KUKA KRL program: MyProgram_101().src

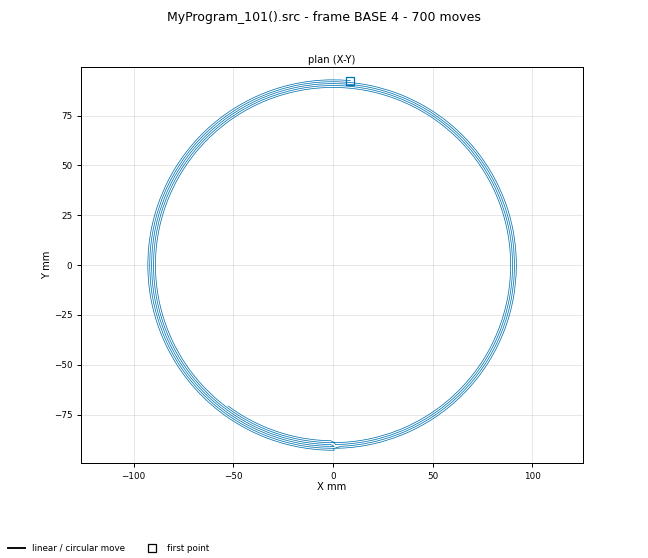
[picture p0: tool path of MyProgram_101().src in frame BASE 4, 700 of 700 moves have a stored position in this frame; points joined in program order, loops and branches not executed]
&ACCESS RVP
&REL 1
&PARAM TEMPLATE = C:\KRC\Roboter\Template\vorgabe
&PARAM EDITMASK = *
DEF MyProgram_101()
; ---- Setting reference (Base) ----
$BASE = BASE_DATA[4]

; --------------------------
; ---- Setting tool (TCP) ----
$TOOL = TOOL_DATA[3]
; --------------------------

$VEL.CP = VEL_APROX_PRINT
Startdeposition()
$VEL.CP = VEL_PRINT
LIN {X 8.6685,Y 92.5128,Z 92,A 80.0856,B 24.9063,C -2.2344,E1 25.0131,E2 4.9435} C_DIS
LIN {X 3.5626,Y 92.8506,Z 92,A 82.8753,B 24.9074,C -2.2219,E1 25.0054,E2 2.1844} C_DIS
LIN {X -2.3592,Y 92.8893,Z 92,A 87.6518,B 24.9042,C -2.2593,E1 24.9918,E2 -2.6809} C_DIS
LIN {X -7.3293,Y 92.6285,Z 92,A 89.5483,B 24.9077,C -2.2184,E1 24.9868,E2 -4.481} C_DIS
LIN {X -9.3778,Y 92.444,Z 92,A 91.7647,B 24.9051,C -2.2495,E1 24.9805,E2 -6.7727} C_DIS
LIN {X -13.6164,Y 91.9165,Z 92,A 93.6976,B 24.9072,C -2.2243,E1 24.9753,E2 -8.6472} C_DIS
LIN {X -16.7897,Y 91.3891,Z 92,A 95.4705,B 24.9079,C -2.2159,E1 24.9704,E2 -10.4018} C_DIS
LIN {X -20.8381,Y 90.5513,Z 92,A 98.1416,B 24.9077,C -2.2177,E1 24.9631,E2 -13.0804} C_DIS
LIN {X -24.0491,Y 89.752,Z 92,A 100.1644,B 24.908,C -2.2151,E1 24.9577,E2 -15.1} C_DIS
LIN {X -27.0285,Y 88.9015,Z 92,A 102.8086,B 24.9061,C -2.2371,E1 24.9504,E2 -17.8011} C_DIS
LIN {X -30.6581,Y 87.7146,Z 92,A 104.1863,B 24.909,C -2.2023,E1 24.947,E2 -19.0985} C_DIS
LIN {X -35.7226,Y 85.7771,Z 92,A 108.0632,B 24.908,C -2.215,E1 24.9368,E2 -23.0141} C_DIS
LIN {X -39.4719,Y 84.1178,Z 92,A 110.5653,B 24.9084,C -2.2103,E1 24.9305,E2 -25.5112} C_DIS
LIN {X -43.093,Y 82.3213,Z 92,A 112.9702,B 24.9089,C -2.2035,E1 24.9245,E2 -27.9061} C_DIS
LIN {X -46.2813,Y 80.5717,Z 92,A 115.1055,B 24.9095,C -2.1961,E1 24.9193,E2 -30.0302} C_DIS
LIN {X -49.1228,Y 78.8715,Z 92,A 116.9389,B 24.9104,C -2.1857,E1 24.915,E2 -31.8445} C_DIS
LIN {X -51.7549,Y 77.1709,Z 92,A 119.2261,B 24.9098,C -2.1933,E1 24.9096,E2 -34.1572} C_DIS
LIN {X -54.5832,Y 75.1969,Z 92,A 121.3196,B 24.9102,C -2.188,E1 24.9049,E2 -36.2452} C_DIS
LIN {X -57.0235,Y 73.3636,Z 92,A 123.1994,B 24.9105,C -2.1839,E1 24.9007,E2 -38.1223} C_DIS
LIN {X -59.5641,Y 71.3156,Z 92,A 124.9102,B 24.9117,C -2.17,E1 24.8971,E2 -39.8064} C_DIS
LIN {X -62.1969,Y 69.0317,Z 92,A 127.4401,B 24.9111,C -2.1772,E1 24.8917,E2 -42.3633} C_DIS
LIN {X -64.7695,Y 66.6245,Z 92,A 129.5058,B 24.9118,C -2.1687,E1 24.8876,E2 -44.4172} C_DIS
LIN {X -66.9884,Y 64.392,Z 92,A 131.5448,B 24.9119,C -2.167,E1 24.8836,E2 -46.4612} C_DIS
LIN {X -68.5485,Y 62.7286,Z 92,A 133.1466,B 24.9117,C -2.1697,E1 24.8805,E2 -48.0763} C_DIS
LIN {X -71.3556,Y 59.516,Z 92,A 135.5018,B 24.913,C -2.1543,E1 24.8763,E2 -50.4056} C_DIS
LIN {X -73.2264,Y 57.2008,Z 92,A 137.5086,B 24.913,C -2.1548,E1 24.8728,E2 -52.423} C_DIS
LIN {X -75.6618,Y 53.9356,Z 92,A 140.3542,B 24.9126,C -2.1585,E1 24.8681,E2 -55.2912} C_DIS
LIN {X -78.3706,Y 49.919,Z 92,A 143.006,B 24.9141,C -2.1396,E1 24.8641,E2 -57.9114} C_DIS
LIN {X -79.8357,Y 47.5405,Z 92,A 145.45,B 24.9127,C -2.1573,E1 24.8605,E2 -60.4101} C_DIS
LIN {X -81.9789,Y 43.7432,Z 92,A 147.2305,B 24.9156,C -2.1211,E1 24.8583,E2 -62.1138} C_DIS
LIN {X -83.9639,Y 39.7993,Z 92,A 150.1955,B 24.9156,C -2.1205,E1 24.8546,E2 -65.0933} C_DIS
LIN {X -86.8415,Y 33.0503,Z 92,A 155.4811,B 24.9149,C -2.1304,E1 24.849,E2 -70.4321} C_DIS
LIN {X -88.3197,Y 28.8698,Z 92,A 157.4147,B 24.9175,C -2.0971,E1 24.8473,E2 -72.297} C_DIS
LIN {X -89.2816,Y 25.7437,Z 92,A 159.2439,B 24.9185,C -2.085,E1 24.8459,E2 -74.1079} C_DIS
LIN {X -90.3116,Y 21.8542,Z 92,A 161.8727,B 24.9187,C -2.0817,E1 24.844,E2 -76.7442} C_DIS
LIN {X -91.0374,Y 18.5998,Z 92,A 163.664,B 24.9199,C -2.0671,E1 24.843,E2 -78.5112} C_DIS
LIN {X -91.5949,Y 15.6278,Z 92,A 166.1987,B 24.9187,C -2.0817,E1 24.8417,E2 -81.0959} C_DIS
LIN {X -92.2271,Y 11.3219,Z 92,A 168.754,B 24.9197,C -2.0691,E1 24.8408,E2 -83.6364} C_DIS
LIN {X -92.6128,Y 7.5252,Z 92,A 171.2761,B 24.9199,C -2.0668,E1 24.8401,E2 -86.1681} C_DIS
LIN {X -92.9096,Y 1.2732,Z 92,A 175.048,B 24.9211,C -2.0517,E1 24.8398,E2 -89.9267} C_DIS
LIN {X -92.8996,Y -1.852,Z 92,A 177.8358,B 24.9195,C -2.0723,E1 24.84,E2 -92.7805} C_DIS
LIN {X -92.65,Y -7.0609,Z 92,A -179.9339,B 24.9226,C -2.0314,E1 24.8404,E2 -94.9264} C_DIS
LIN {X -92.3349,Y -10.401,Z 92,A -177.8054,B 24.923,C -2.0267,E1 24.841,E2 -97.0564} C_DIS
LIN {X -91.8721,Y -13.905,Z 92,A -175.6926,B 24.9237,C -2.0178,E1 24.8418,E2 -99.1606} C_DIS
LIN {X -91.3402,Y -17.0584,Z 92,A -173.6234,B 24.9239,C -2.0146,E1 24.8428,E2 -101.2346} C_DIS
LIN {X -90.635,Y -20.4756,Z 92,A -171.7293,B 24.925,C -2,E1 24.8439,E2 -103.105} C_DIS
LIN {X -89.8976,Y -23.5016,Z 92,A -168.9165,B 24.9233,C -2.022,E1 24.8459,E2 -105.9866} C_DIS
LIN {X -88.8201,Y -27.2909,Z 92,A -167.1243,B 24.9254,C -1.9947,E1 24.8473,E2 -107.7241} C_DIS
LIN {X -87.6746,Y -30.7721,Z 92,A -164.9819,B 24.9262,C -1.9844,E1 24.8492,E2 -109.854} C_DIS
LIN {X -86.4825,Y -33.9783,Z 92,A -162.2464,B 24.9252,C -1.9979,E1 24.852,E2 -112.6371} C_DIS
LIN {X -85.1973,Y -37.0834,Z 92,A -160.6883,B 24.9268,C -1.9758,E1 24.8537,E2 -114.1511} C_DIS
LIN {X -83.8317,Y -40.0753,Z 92,A -158.6212,B 24.9271,C -1.9713,E1 24.8562,E2 -116.2188} C_DIS
LIN {X -82.2602,Y -43.2091,Z 92,A -156.425,B 24.9275,C -1.9664,E1 24.859,E2 -118.4152} C_DIS
LIN {X -79.7757,Y -47.6421,Z 92,A -153.2654,B 24.9281,C -1.9589,E1 24.8633,E2 -121.5731} C_DIS
LIN {X -77.3395,Y -51.5028,Z 92,A -150.4483,B 24.9286,C -1.9517,E1 24.8676,E2 -124.3874} C_DIS
LIN {X -74.9207,Y -54.9604,Z 92,A -147.9325,B 24.9293,C -1.9425,E1 24.8717,E2 -126.8935} C_DIS
LIN {X -72.9573,Y -57.5411,Z 92,A -145.9634,B 24.9297,C -1.9367,E1 24.875,E2 -128.8583} C_DIS
LIN {X -70.924,Y -60.0302,Z 92,A -143.3889,B 24.9286,C -1.9511,E1 24.8797,E2 -131.4788} C_DIS
LIN {X -68.7858,Y -62.47,Z 92,A -141.7905,B 24.9299,C -1.9337,E1 24.8826,E2 -133.0429} C_DIS
LIN {X -67.1259,Y -64.2492,Z 92,A -139.9944,B 24.9294,C -1.94,E1 24.8861,E2 -134.8618} C_DIS
LIN {X -63.1282,Y -68.1818,Z 92,A -136.838,B 24.9307,C -1.9231,E1 24.8924,E2 -137.991} C_DIS
LIN {X -60.9567,Y -70.1291,Z 92,A -135.1059,B 24.9311,C -1.9175,E1 24.8961,E2 -139.7165} C_DIS
LIN {X -58.2775,Y -72.3711,Z 92,A -132.4598,B 24.9302,C -1.9295,E1 24.9019,E2 -142.4012} C_DIS
LIN {X -54.9904,Y -74.8987,Z 92,A -130.2116,B 24.9313,C -1.9149,E1 24.9068,E2 -144.6228} C_DIS
LIN {X -51.8971,Y -77.0746,Z 92,A -128.2718,B 24.9324,C -1.8983,E1 24.9112,E2 -146.5296} C_DIS
LIN {X -49.5179,Y -78.6247,Z 92,A -126.3962,B 24.9324,C -1.8996,E1 24.9156,E2 -148.4145} C_DIS
LIN {X -44.9776,Y -81.3062,Z 92,A -122.7756,B 24.9318,C -1.9072,E1 24.9245,E2 -152.0639} C_DIS
LIN {X -40.832,Y -83.467,Z 92,A -119.7997,B 24.9318,C -1.9067,E1 24.9319,E2 -155.0464} C_DIS
LIN {X -36.8853,Y -85.2837,Z 92,A -117.4804,B 24.9329,C -1.8918,E1 24.9377,E2 -157.3359} C_DIS
LIN {X -33.9003,Y -86.5132,Z 92,A -115.3671,B 24.9328,C -1.8939,E1 24.9432,E2 -159.4589} C_DIS
LIN {X -30.6688,Y -87.7108,Z 92,A -112.9272,B 24.9321,C -1.9027,E1 24.9497,E2 -161.9245} C_DIS
LIN {X -26.0912,Y -89.1803,Z 92,A -110.4074,B 24.9334,C -1.8855,E1 24.9563,E2 -164.4077} C_DIS
LIN {X -22.9049,Y -90.0509,Z 92,A -107.9771,B 24.9325,C -1.8976,E1 24.963,E2 -166.8706} C_DIS
LIN {X -18.0534,Y -91.1486,Z 92,A -105.1442,B 24.9332,C -1.8882,E1 24.9707,E2 -169.6846} C_DIS
LIN {X -12.8895,Y -92.0198,Z 92,A -102.102,B 24.9337,C -1.8809,E1 24.979,E2 -172.7123} C_DIS
LIN {X -8.1132,Y -92.5641,Z 92,A -98.9097,B 24.9331,C -1.8884,E1 24.9879,E2 -175.9242} C_DIS
LIN {X -5.2842,Y -92.7677,Z 92,A -96.7874,B 24.9322,C -1.9014,E1 24.9939,E2 -178.0781} C_DIS
LIN {X -2.0857,Y -92.8953,Z 92,A -95.1973,B 24.9332,C -1.8884,E1 24.9983,E2 -179.6373} C_DIS
LIN {X 0.616,Y -92.9061,Z 92,A -93.7308,B 24.9336,C -1.882,E1 25.0024,E2 -181.0887} C_DIS
Enddeposition()
LIN {X 0.616,Y -92.9061,Z 92,A -93.7308,B 24.9336,C -1.882,E1 25.0024,E2 -181.0887} C_DIS
Startdeposition()
$VEL.CP = VEL_PRINT
LIN {X 0.2828,Y -91.9616,Z 92,A -94.5574,B 24.9339,C -1.8772,E1 25,E2 -180.2507} C_DIS
LIN {X -5.5997,Y -91.7928,Z 92,A -98.2442,B 24.934,C -1.876,E1 24.9897,E2 -176.5604} C_DIS
LIN {X -11.5025,Y -91.2403,Z 92,A -102.7915,B 24.936,C -1.848,E1 24.9769,E2 -171.9441} C_DIS
LIN {X -15.3961,Y -90.6643,Z 92,A -104.5195,B 24.9343,C -1.8726,E1 24.9723,E2 -170.273} C_DIS
LIN {X -18.6363,Y -90.0539,Z 92,A -107.2484,B 24.9358,C -1.8513,E1 24.9647,E2 -167.4902} C_DIS
LIN {X -22.3727,Y -89.2006,Z 92,A -108.8615,B 24.9339,C -1.8779,E1 24.9605,E2 -165.9382} C_DIS
LIN {X -24.9821,Y -88.5037,Z 92,A -110.8484,B 24.9345,C -1.869,E1 24.955,E2 -163.927} C_DIS
LIN {X -27.644,Y -87.7097,Z 92,A -113.1828,B 24.9358,C -1.8507,E1 24.9487,E2 -161.545} C_DIS
LIN {X -31.573,Y -86.3721,Z 92,A -114.7673,B 24.9334,C -1.8854,E1 24.9448,E2 -160.0398} C_DIS
LIN {X -33.8196,Y -85.5177,Z 92,A -116.5155,B 24.9338,C -1.8786,E1 24.9401,E2 -158.2718} C_DIS
LIN {X -37.183,Y -84.1109,Z 92,A -119.0663,B 24.9343,C -1.872,E1 24.9335,E2 -155.6992} C_DIS
LIN {X -40.4944,Y -82.5672,Z 92,A -121.1125,B 24.9336,C -1.8821,E1 24.9284,E2 -153.6718} C_DIS
LIN {X -43.5278,Y -81.009,Z 92,A -123.807,B 24.9347,C -1.8667,E1 24.9217,E2 -150.9332} C_DIS
LIN {X -46.6784,Y -79.2347,Z 92,A -125.4312,B 24.933,C -1.8899,E1 24.9179,E2 -149.3592} C_DIS
LIN {X -48.8539,Y -77.9122,Z 92,A -127.4045,B 24.9337,C -1.8799,E1 24.9131,E2 -147.3561} C_DIS
LIN {X -51.7207,Y -76.0395,Z 92,A -129.5924,B 24.9337,C -1.8816,E1 24.9081,E2 -145.1649} C_DIS
LIN {X -55.1728,Y -73.5728,Z 92,A -132.7055,B 24.9343,C -1.8716,E1 24.901,E2 -142.0168} C_DIS
LIN {X -58.7179,Y -70.7758,Z 92,A -134.2641,B 24.9312,C -1.916,E1 24.8979,E2 -140.5582} C_DIS
LIN {X -60.4642,Y -69.2898,Z 92,A -136.1318,B 24.932,C -1.9049,E1 24.8938,E2 -138.6567} C_DIS
LIN {X -64.9463,Y -65.1083,Z 92,A -140.1141,B 24.9318,C -1.9076,E1 24.8858,E2 -134.6645} C_DIS
LIN {X -67.8507,Y -62.0749,Z 92,A -143.4197,B 24.9329,C -1.8922,E1 24.8794,E2 -131.3075} C_DIS
LIN {X -70.7868,Y -58.7047,Z 92,A -144.8676,B 24.9295,C -1.9398,E1 24.877,E2 -129.9665} C_DIS
LIN {X -73.1722,Y -55.7055,Z 92,A -148.3649,B 24.9315,C -1.9113,E1 24.8708,E2 -126.3846} C_DIS
LIN {X -75.2745,Y -52.8291,Z 92,A -149.7922,B 24.9294,C -1.9411,E1 24.8686,E2 -125.0214} C_DIS
LIN {X -76.6509,Y -50.8103,Z 92,A -152.1221,B 24.9309,C -1.9203,E1 24.8649,E2 -122.6302} C_DIS
LIN {X -78.5609,Y -47.8035,Z 92,A -154.4332,B 24.9307,C -1.9233,E1 24.8615,E2 -120.3145} C_DIS
LIN {X -80.5191,Y -44.4285,Z 92,A -155.9549,B 24.9282,C -1.9574,E1 24.8596,E2 -118.8662} C_DIS
LIN {X -82.2624,Y -41.1094,Z 92,A -158.5863,B 24.9284,C -1.9548,E1 24.8561,E2 -116.2145} C_DIS
LIN {X -83.5972,Y -38.3248,Z 92,A -160.6338,B 24.9282,C -1.9565,E1 24.8537,E2 -114.1598} C_DIS
LIN {X -85.0169,Y -35.0606,Z 92,A -163.1255,B 24.9284,C -1.9546,E1 24.851,E2 -111.6498} C_DIS
LIN {X -87.0622,Y -29.6179,Z 92,A -166.3552,B 24.9267,C -1.9771,E1 24.848,E2 -108.4554} C_DIS
LIN {X -88.9962,Y -23.1677,Z 92,A -170.3149,B 24.9252,C -1.9968,E1 24.8449,E2 -104.52} C_DIS
LIN {X -89.9931,Y -18.9325,Z 92,A -173.4017,B 24.9255,C -1.9938,E1 24.8429,E2 -101.4079} C_DIS
LIN {X -90.6389,Y -15.5479,Z 92,A -175.5804,B 24.925,C -1.9995,E1 24.8418,E2 -99.2299} C_DIS
LIN {X -91.1795,Y -11.9711,Z 92,A -177.8201,B 24.9245,C -2.007,E1 24.841,E2 -96.9948} C_DIS
LIN {X -91.5934,Y -8.2281,Z 92,A 179.8874,B 24.9238,C -2.0161,E1 24.8403,E2 -94.71} C_DIS
LIN {X -91.9262,Y -2.5761,Z 92,A 176.4109,B 24.9228,C -2.0288,E1 24.8398,E2 -91.2431} C_DIS
LIN {X -91.9611,Y 0.452,Z 92,A 173.6815,B 24.9243,C -2.0099,E1 24.8398,E2 -88.4521} C_DIS
LIN {X -91.8509,Y 4.5052,Z 92,A 171.9899,B 24.9218,C -2.0427,E1 24.84,E2 -86.8287} C_DIS
LIN {X -91.7204,Y 6.6768,Z 92,A 170.4237,B 24.9219,C -2.0407,E1 24.8403,E2 -85.2484} C_DIS
LIN {X -91.3851,Y 10.292,Z 92,A 168.0913,B 24.9215,C -2.0459,E1 24.841,E2 -82.9142} C_DIS
LIN {X -90.947,Y 13.6316,Z 92,A 165.9194,B 24.9212,C -2.0504,E1 24.8419,E2 -80.7403} C_DIS
LIN {X -90.2374,Y 17.7291,Z 92,A 163.7941,B 24.9194,C -2.0726,E1 24.8429,E2 -78.6551} C_DIS
LIN {X -89.3345,Y 21.8254,Z 92,A 159.9783,B 24.9216,C -2.0453,E1 24.8454,E2 -74.7518} C_DIS
LIN {X -88.1157,Y 26.3181,Z 92,A 158.5099,B 24.9175,C -2.0969,E1 24.8464,E2 -73.3981} C_DIS
LIN {X -85.8343,Y 33.0105,Z 92,A 153.8445,B 24.9171,C -2.1026,E1 24.8506,E2 -68.7199} C_DIS
LIN {X -83.9426,Y 37.5591,Z 92,A 150.096,B 24.918,C -2.0916,E1 24.8548,E2 -64.9242} C_DIS
LIN {X -81.4075,Y 42.7764,Z 92,A 146.5129,B 24.917,C -2.1032,E1 24.8593,E2 -61.3495} C_DIS
LIN {X -78.8588,Y 47.3134,Z 92,A 143.6783,B 24.9153,C -2.1247,E1 24.8632,E2 -58.5515} C_DIS
LIN {X -75.1466,Y 53.0116,Z 92,A 138.8684,B 24.9158,C -2.1193,E1 24.8707,E2 -53.7046} C_DIS
LIN {X -72.4594,Y 56.6294,Z 92,A 136.3327,B 24.9145,C -2.1349,E1 24.8749,E2 -51.1942} C_DIS
LIN {X -70.1399,Y 59.4763,Z 92,A 133.514,B 24.9153,C -2.1249,E1 24.88,E2 -48.3386} C_DIS
LIN {X -67.6898,Y 62.2503,Z 92,A 131.9427,B 24.9131,C -2.1529,E1 24.8829,E2 -46.827} C_DIS
LIN {X -65.6704,Y 64.3779,Z 92,A 129.8996,B 24.9132,C -2.1507,E1 24.8869,E2 -44.77} C_DIS
LIN {X -63.0701,Y 66.9266,Z 92,A 127.6993,B 24.9126,C -2.1582,E1 24.8913,E2 -42.5783} C_DIS
LIN {X -58.7476,Y 70.7511,Z 92,A 124.1726,B 24.9118,C -2.1684,E1 24.8987,E2 -39.0621} C_DIS
LIN {X -56.3635,Y 72.6652,Z 92,A 122.0966,B 24.9119,C -2.1672,E1 24.9032,E2 -36.9756} C_DIS
LIN {X -53.4043,Y 74.8664,Z 92,A 119.5836,B 24.9121,C -2.1653,E1 24.9089,E2 -34.4492} C_DIS
LIN {X -48.3848,Y 78.2053,Z 92,A 116.0419,B 24.9109,C -2.1791,E1 24.9172,E2 -30.9289} C_DIS
LIN {X -45.5415,Y 79.8941,Z 92,A 113.9873,B 24.9106,C -2.1829,E1 24.9221,E2 -28.8773} C_DIS
LIN {X -41.9369,Y 81.8432,Z 92,A 110.8076,B 24.9119,C -2.1677,E1 24.9301,E2 -25.6527} C_DIS
LIN {X -38.4781,Y 83.5258,Z 92,A 109.4852,B 24.9088,C -2.205,E1 24.9333,E2 -24.4156} C_DIS
LIN {X -32.1419,Y 86.1632,Z 92,A 104.9607,B 24.909,C -2.2031,E1 24.945,E2 -19.8763} C_DIS
LIN {X -26.3547,Y 88.1049,Z 92,A 101.0991,B 24.9087,C -2.2057,E1 24.9552,E2 -16.0139} C_DIS
LIN {X -23.8607,Y 88.8126,Z 92,A 99.4038,B 24.9088,C -2.2048,E1 24.9598,E2 -14.3139} C_DIS
LIN {X -19.4825,Y 89.8746,Z 92,A 96.4999,B 24.9088,C -2.2043,E1 24.9677,E2 -11.4049} C_DIS
LIN {X -16.833,Y 90.41,Z 92,A 94.7575,B 24.9089,C -2.2038,E1 24.9725,E2 -9.6592} C_DIS
LIN {X -13.905,Y 90.9047,Z 92,A 92.9109,B 24.9088,C -2.2052,E1 24.9776,E2 -7.8144} C_DIS
LIN {X -9.4125,Y 91.4791,Z 92,A 90.4784,B 24.9076,C -2.2195,E1 24.9842,E2 -5.414} C_DIS
LIN {X -7.0352,Y 91.6929,Z 92,A 87.9373,B 24.9104,C -2.1859,E1 24.9915,E2 -2.7923} C_DIS
LIN {X -2.9739,Y 91.9139,Z 92,A 86.3341,B 24.9078,C -2.217,E1 24.9958,E2 -1.2625} C_DIS
LIN {X 1.9013,Y 91.9425,Z 92,A 83.2214,B 24.908,C -2.2151,E1 25.0045,E2 1.8546} C_DIS
LIN {X 8.2335,Y 91.5929,Z 92,A 79.4639,B 24.9074,C -2.2215,E1 25.0149,E2 5.5954} C_DIS
LIN {X 12.3597,Y 91.1292,Z 92,A 76.4373,B 24.9087,C -2.2064,E1 25.0234,E2 8.6557} C_DIS
LIN {X 15.7547,Y 90.6039,Z 92,A 73.6994,B 24.9104,C -2.1858,E1 25.0311,E2 11.4394} C_DIS
LIN {X 19.649,Y 89.8383,Z 92,A 71.9868,B 24.9084,C -2.21,E1 25.0356,E2 13.0925} C_DIS
LIN {X 22.2254,Y 89.2369,Z 92,A 70.0924,B 24.9091,C -2.2008,E1 25.0408,E2 15.0061} C_DIS
LIN {X 28.415,Y 87.4619,Z 92,A 66.2333,B 24.909,C -2.203,E1 25.0511,E2 18.8531} C_DIS
LIN {X 31.8114,Y 86.2852,Z 92,A 63.9048,B 24.9094,C -2.198,E1 25.0572,E2 21.1888} C_DIS
LIN {X 34.3944,Y 85.2884,Z 92,A 61.9301,B 24.9102,C -2.1878,E1 25.0624,E2 23.1831} C_DIS
LIN {X 38.7426,Y 83.4027,Z 92,A 59.388,B 24.9093,C -2.1985,E1 25.0688,E2 25.6937} C_DIS
LIN {X 43.4952,Y 81.0255,Z 92,A 56.0505,B 24.9098,C -2.1933,E1 25.0771,E2 29.0342} C_DIS
LIN {X 46.2149,Y 79.5072,Z 92,A 53.7973,B 24.9109,C -2.1797,E1 25.0826,E2 31.3127} C_DIS
LIN {X 49.9134,Y 77.2381,Z 92,A 51.2644,B 24.9107,C -2.1815,E1 25.0885,E2 33.8334} C_DIS
LIN {X 52.3849,Y 75.5833,Z 92,A 49.0162,B 24.9121,C -2.1647,E1 25.0938,E2 36.1135} C_DIS
LIN {X 55.3268,Y 73.4571,Z 92,A 46.7079,B 24.9126,C -2.1591,E1 25.0989,E2 38.4268} C_DIS
LIN {X 58.3824,Y 71.0545,Z 92,A 45.1022,B 24.9106,C -2.1831,E1 25.1023,E2 39.9698} C_DIS
LIN {X 60.6518,Y 69.126,Z 92,A 43.0142,B 24.9116,C -2.1713,E1 25.1067,E2 42.0775} C_DIS
LIN {X 63.6497,Y 66.3759,Z 92,A 40.7956,B 24.9111,C -2.1773,E1 25.1112,E2 44.2728} C_DIS
LIN {X 65.3279,Y 64.7246,Z 92,A 39.0883,B 24.912,C -2.1657,E1 25.1146,E2 46.0004} C_DIS
LIN {X 68.0138,Y 61.8971,Z 92,A 36.3554,B 24.9133,C -2.1496,E1 25.1199,E2 48.7594} C_DIS
LIN {X 70.6202,Y 58.905,Z 92,A 34.2149,B 24.9128,C -2.1556,E1 25.1237,E2 50.8758} C_DIS
LIN {X 73.0518,Y 55.8618,Z 92,A 32.0135,B 24.9127,C -2.1579,E1 25.1275,E2 53.0615} C_DIS
LIN {X 74.5764,Y 53.8107,Z 92,A 29.9752,B 24.9143,C -2.138,E1 25.1309,E2 55.137} C_DIS
LIN {X 77.6741,Y 49.2342,Z 92,A 26.6174,B 24.9147,C -2.1322,E1 25.1361,E2 58.4917} C_DIS
LIN {X 79.6578,Y 45.9528,Z 92,A 24.4327,B 24.9147,C -2.1332,E1 25.1391,E2 60.6628} C_DIS
LIN {X 81.5998,Y 42.4112,Z 92,A 21.7393,B 24.9157,C -2.12,E1 25.1427,E2 63.3733} C_DIS
LIN {X 83.0177,Y 39.562,Z 92,A 19.7845,B 24.9161,C -2.1154,E1 25.1451,E2 65.3283} C_DIS
LIN {X 85.2013,Y 34.6083,Z 92,A 16.157,B 24.9176,C -2.0966,E1 25.1491,E2 68.9804} C_DIS
LIN {X 86.6592,Y 30.7781,Z 92,A 14.0219,B 24.917,C -2.1042,E1 25.1511,E2 71.0856} C_DIS
LIN {X 87.8023,Y 27.3453,Z 92,A 11.6532,B 24.9178,C -2.0933,E1 25.1531,E2 73.4666} C_DIS
LIN {X 88.6607,Y 24.4231,Z 92,A 9.9022,B 24.9178,C -2.0929,E1 25.1545,E2 75.2086} C_DIS
LIN {X 89.8415,Y 19.634,Z 92,A 6.2087,B 24.9204,C -2.0609,E1 25.1568,E2 78.9561} C_DIS
LIN {X 90.6181,Y 15.6721,Z 92,A 4.555,B 24.9185,C -2.0844,E1 25.1576,E2 80.5446} C_DIS
LIN {X 91.4737,Y 9.4642,Z 92,A 0.6816,B 24.9194,C -2.0732,E1 25.159,E2 84.4215} C_DIS
LIN {X 91.8931,Y 3.5759,Z 92,A -2.9164,B 24.9201,C -2.0644,E1 25.1597,E2 88.019} C_DIS
LIN {X 91.9585,Y -0.8351,Z 92,A -5.8986,B 24.9214,C -2.047,E1 25.1597,E2 91.0245} C_DIS
LIN {X 91.8212,Y -5.0846,Z 92,A -8.9068,B 24.9231,C -2.0254,E1 25.1594,E2 94.0658} C_DIS
LIN {X 91.0208,Y -13.1238,Z 92,A -13.9681,B 24.9244,C -2.0082,E1 25.1577,E2 99.1377} C_DIS
LIN {X 90.5052,Y -16.3037,Z 92,A -15.455,B 24.9234,C -2.0208,E1 25.157,E2 100.5861} C_DIS
LIN {X 89.5013,Y -21.1332,Z 92,A -18.4839,B 24.924,C -2.0127,E1 25.1553,E2 103.6167} C_DIS
LIN {X 88.4836,Y -25.053,Z 92,A -21.0539,B 24.9248,C -2.003,E1 25.1534,E2 106.1947} C_DIS
LIN {X 87.4607,Y -28.4189,Z 92,A -23.724,B 24.9266,C -1.9787,E1 25.1511,E2 108.9071} C_DIS
LIN {X 86.3759,Y -31.5628,Z 92,A -24.797,B 24.9243,C -2.0089,E1 25.1502,E2 109.9028} C_DIS
LIN {X 85.1636,Y -34.701,Z 92,A -27.7218,B 24.9271,C -1.972,E1 25.1471,E2 112.8983} C_DIS
LIN {X 83.6955,Y -38.1075,Z 92,A -29.7485,B 24.9268,C -1.9754,E1 25.1448,E2 114.9061} C_DIS
LIN {X 81.3991,Y -42.7923,Z 92,A -32.6428,B 24.9266,C -1.9788,E1 25.1413,E2 117.777} C_DIS
LIN {X 79.0732,Y -46.9517,Z 92,A -35.8269,B 24.9278,C -1.9623,E1 25.1368,E2 120.9834} C_DIS
LIN {X 77.3233,Y -49.7808,Z 92,A -37.8365,B 24.9281,C -1.9587,E1 25.1338,E2 122.9914} C_DIS
LIN {X 75.5907,Y -52.3742,Z 92,A -39.8359,B 24.9286,C -1.9513,E1 25.1307,E2 124.9985} C_DIS
LIN {X 73.5566,Y -55.1944,Z 92,A -42.5624,B 24.9305,C -1.9251,E1 25.1261,E2 127.7736} C_DIS
LIN {X 71.339,Y -58.0325,Z 92,A -44.9739,B 24.9314,C -1.9132,E1 25.1218,E2 130.202} C_DIS
LIN {X 68.6019,Y -61.2437,Z 92,A -46.4496,B 24.9289,C -1.9481,E1 25.1193,E2 131.5888} C_DIS
LIN {X 66.9912,Y -63.0014,Z 92,A -49.0653,B 24.9321,C -1.9037,E1 25.1141,E2 134.2979} C_DIS
LIN {X 64.0171,Y -66.0218,Z 92,A -51.6536,B 24.9324,C -1.8992,E1 25.1089,E2 136.886} C_DIS
LIN {X 60.9981,Y -68.8217,Z 92,A -53.3271,B 24.9305,C -1.9251,E1 25.1056,E2 138.4916} C_DIS
LIN {X 59.1259,Y -70.4368,Z 92,A -55.7994,B 24.9331,C -1.8884,E1 25.1001,E2 141.041} C_DIS
LIN {X 55.7736,Y -73.1198,Z 92,A -58.1721,B 24.9328,C -1.8934,E1 25.0949,E2 143.3933} C_DIS
LIN {X 53.1514,Y -75.0468,Z 92,A -59.5537,B 24.9315,C -1.9122,E1 25.0919,E2 144.7257} C_DIS
LIN {X 50.879,Y -76.6056,Z 92,A -61.4423,B 24.9321,C -1.9027,E1 25.0875,E2 146.6304} C_DIS
LIN {X 48.0906,Y -78.3864,Z 92,A -63.8762,B 24.9333,C -1.8856,E1 25.0816,E2 149.0969} C_DIS
LIN {X 44.6891,Y -80.3735,Z 92,A -65.7662,B 24.9322,C -1.9011,E1 25.0771,E2 150.9445} C_DIS
LIN {X 42.1864,Y -81.7156,Z 92,A -68.261,B 24.9343,C -1.8726,E1 25.0708,E2 153.4998} C_DIS
LIN {X 38.955,Y -83.3038,Z 92,A -70.3855,B 24.9343,C -1.8733,E1 25.0654,E2 155.6174} C_DIS
LIN {X 35.9751,Y -84.6337,Z 92,A -71.6419,B 24.9325,C -1.8974,E1 25.0624,E2 156.8136} C_DIS
LIN {X 30.368,Y -86.8032,Z 92,A -75.9565,B 24.9343,C -1.8725,E1 25.051,E2 161.1779} C_DIS
LIN {X 24.4935,Y -88.6416,Z 92,A -79.3437,B 24.9335,C -1.8836,E1 25.042,E2 164.5328} C_DIS
LIN {X 20.2855,Y -89.6977,Z 92,A -82.3055,B 24.9343,C -1.872,E1 25.0339,E2 167.5178} C_DIS
LIN {X 16.8181,Y -90.4126,Z 92,A -84.2959,B 24.9339,C -1.8776,E1 25.0285,E2 169.4927} C_DIS
LIN {X 13.945,Y -90.8985,Z 92,A -86.7745,B 24.9356,C -1.8536,E1 25.0215,E2 172.0256} C_DIS
LIN {X 10.4021,Y -91.3722,Z 92,A -88.3174,B 24.9341,C -1.8755,E1 25.0174,E2 173.5154} C_DIS
LIN {X 5.3436,Y -91.8069,Z 92,A -91.2893,B 24.9337,C -1.8805,E1 25.0092,E2 176.474} C_DIS
LIN {X 0.5912,Y -91.9536,Z 92,A -93.06,B 24.9309,C -1.9205,E1 25.0046,E2 178.1492} C_DIS
Enddeposition()
LIN {X 0.5912,Y -91.9536,Z 92,A -93.06,B 24.9309,C -1.9205,E1 25.0046,E2 178.1492} C_DIS
Startdeposition()
$VEL.CP = VEL_PRINT
LIN {X 4.0889,Y -90.9141,Z 92,A -91.4298,B 24.931,C -1.9178,E1 25.009,E2 176.5259} C_DIS
LIN {X 7.1118,Y -90.7277,Z 92,A -89.5434,B 24.931,C -1.918,E1 25.0143,E2 174.64} C_DIS
LIN {X 11.0267,Y -90.3358,Z 92,A -86.7492,B 24.9301,C -1.9304,E1 25.0221,E2 171.8184} C_DIS
LIN {X 15.4148,Y -89.6918,Z 92,A -84.224,B 24.9307,C -1.9232,E1 25.029,E2 169.3128} C_DIS
LIN {X 18.7307,Y -89.0585,Z 92,A -81.8883,B 24.93,C -1.9323,E1 25.0354,E2 166.9583} C_DIS
LIN {X 22.6976,Y -88.1299,Z 92,A -79.7337,B 24.9308,C -1.9206,E1 25.0412,E2 164.8347} C_DIS
LIN {X 28.3671,Y -86.4726,Z 92,A -76.0286,B 24.9306,C -1.9243,E1 25.0511,E2 161.1274} C_DIS
LIN {X 33.2291,Y -84.7224,Z 92,A -72.5336,B 24.9297,C -1.9371,E1 25.0603,E2 157.6094} C_DIS
LIN {X 35.9929,Y -83.5867,Z 92,A -69.4735,B 24.9264,C -1.9819,E1 25.0684,E2 154.4506} C_DIS
LIN {X 41.4959,Y -80.9948,Z 92,A -66.8827,B 24.9292,C -1.9438,E1 25.0746,E2 151.957} C_DIS
LIN {X 43.7943,Y -79.7768,Z 92,A -64.4746,B 24.9269,C -1.9742,E1 25.0807,E2 149.484} C_DIS
LIN {X 47.7526,Y -77.4729,Z 92,A -62.381,B 24.9286,C -1.9511,E1 25.0855,E2 147.4514} C_DIS
LIN {X 50.6673,Y -75.5981,Z 92,A -60.2052,B 24.9283,C -1.9552,E1 25.0906,E2 145.2733} C_DIS
LIN {X 53.3211,Y -73.7511,Z 92,A -57.9909,B 24.9275,C -1.9658,E1 25.0957,E2 143.0416} C_DIS
LIN {X 57.8514,Y -70.2527,Z 92,A -54.6385,B 24.9276,C -1.9645,E1 25.103,E2 139.7046} C_DIS
LIN {X 60.4872,Y -67.9959,Z 92,A -52.6353,B 24.9278,C -1.963,E1 25.1072,E2 137.713} C_DIS
LIN {X 63.6055,Y -65.0896,Z 92,A -49.341,B 24.9256,C -1.9915,E1 25.1139,E2 134.365} C_DIS
LIN {X 65.9276,Y -62.7368,Z 92,A -47.6882,B 24.9264,C -1.981,E1 25.1171,E2 132.7441} C_DIS
LIN {X 68.2977,Y -60.1468,Z 92,A -45.8094,B 24.9269,C -1.9746,E1 25.1205,E2 130.8887} C_DIS
LIN {X 70.792,Y -57.189,Z 92,A -42.7931,B 24.9248,C -2.0021,E1 25.126,E2 127.8214} C_DIS
LIN {X 73.647,Y -53.4633,Z 92,A -40.1528,B 24.9251,C -1.9986,E1 25.1304,E2 125.202} C_DIS
LIN {X 75.6072,Y -50.6538,Z 92,A -37.9548,B 24.9245,C -2.0061,E1 25.1338,E2 122.9973} C_DIS
LIN {X 77.5721,Y -47.5898,Z 92,A -35.9516,B 24.9248,C -2.002,E1 25.1368,E2 121.0138} C_DIS
LIN {X 78.7192,Y -45.6671,Z 92,A -33.7958,B 24.9225,C -2.0336,E1 25.1399,E2 118.7946} C_DIS
LIN {X 80.4573,Y -42.5288,Z 92,A -31.4886,B 24.9218,C -2.042,E1 25.1429,E2 116.4796} C_DIS
LIN {X 82.1938,Y -39.069,Z 92,A -29.7158,B 24.9231,C -2.0247,E1 25.145,E2 114.7571} C_DIS
LIN {X 83.2065,Y -36.8648,Z 92,A -27.1306,B 24.9198,C -2.0686,E1 25.148,E2 112.0826} C_DIS
LIN {X 85.192,Y -32.0069,Z 92,A -25.5174,B 24.9238,C -2.0162,E1 25.1495,E2 110.602} C_DIS
LIN {X 86.69,Y -27.6951,Z 92,A -22.0075,B 24.9213,C -2.0484,E1 25.1527,E2 107.0358} C_DIS
LIN {X 87.432,Y -25.2574,Z 92,A -20.0533,B 24.9199,C -2.0663,E1 25.1543,E2 105.0505} C_DIS
LIN {X 88.373,Y -21.7325,Z 92,A -17.6187,B 24.919,C -2.0787,E1 25.1559,E2 102.6006} C_DIS
LIN {X 89.1538,Y -18.2665,Z 92,A -15.9697,B 24.9201,C -2.064,E1 25.1568,E2 100.996} C_DIS
LIN {X 89.6825,Y -15.4705,Z 92,A -13.9298,B 24.9189,C -2.0789,E1 25.1578,E2 98.9328} C_DIS
LIN {X 90.5655,Y -8.9565,Z 92,A -10.0396,B 24.9186,C -2.083,E1 25.1592,E2 95.056} C_DIS
LIN {X 90.7781,Y -6.442,Z 92,A -7.8966,B 24.9166,C -2.1087,E1 25.1596,E2 92.8651} C_DIS
LIN {X 90.9629,Y -2.7958,Z 92,A -6.198,B 24.9178,C -2.0938,E1 25.1598,E2 91.2118} C_DIS
LIN {X 90.9773,Y 2.328,Z 92,A -2.945,B 24.9169,C -2.1051,E1 25.1597,E2 87.9515} C_DIS
LIN {X 90.6145,Y 8.4312,Z 92,A 0.3099,B 24.9176,C -2.0955,E1 25.1591,E2 84.7384} C_DIS
LIN {X 90.1396,Y 12.5298,Z 92,A 3.3549,B 24.9157,C -2.1201,E1 25.1581,E2 81.6535} C_DIS
LIN {X 89.6348,Y 15.7419,Z 92,A 5.1777,B 24.9158,C -2.1182,E1 25.1573,E2 79.8458} C_DIS
LIN {X 88.8806,Y 19.5531,Z 92,A 8.1185,B 24.9138,C -2.144,E1 25.1556,E2 76.8613} C_DIS
LIN {X 87.8792,Y 23.6498,Z 92,A 10.4875,B 24.914,C -2.1416,E1 25.1539,E2 74.5117} C_DIS
LIN {X 86.5175,Y 28.2284,Z 92,A 13.5636,B 24.9131,C -2.1531,E1 25.1514,E2 71.4259} C_DIS
LIN {X 85.6258,Y 30.829,Z 92,A 15.9552,B 24.9107,C -2.1825,E1 25.1491,E2 68.9784} C_DIS
LIN {X 84.1007,Y 34.7763,Z 92,A 18.5421,B 24.9103,C -2.1873,E1 25.1463,E2 66.3943} C_DIS
LIN {X 82.5188,Y 38.3759,Z 92,A 20.2715,B 24.9119,C -2.167,E1 25.1444,E2 64.7222} C_DIS
LIN {X 81.2799,Y 40.9382,Z 92,A 22.5783,B 24.91,C -2.1907,E1 25.1414,E2 62.3717} C_DIS
LIN {X 79.7525,Y 43.839,Z 92,A 24.2243,B 24.9108,C -2.1811,E1 25.1393,E2 60.757} C_DIS
LIN {X 78.0224,Y 46.8488,Z 92,A 26.1366,B 24.9111,C -2.177,E1 25.1366,E2 58.8642} C_DIS
LIN {X 76.6997,Y 48.9822,Z 92,A 27.8851,B 24.9103,C -2.1872,E1 25.134,E2 57.1004} C_DIS
LIN {X 74.1284,Y 52.7926,Z 92,A 30.7477,B 24.9098,C -2.1934,E1 25.1295,E2 54.2373} C_DIS
LIN {X 72.0309,Y 55.6203,Z 92,A 32.7592,B 24.9099,C -2.1914,E1 25.1261,E2 52.2401} C_DIS
LIN {X 70.2232,Y 57.887,Z 92,A 34.8185,B 24.9089,C -2.2041,E1 25.1224,E2 50.1603} C_DIS
LIN {X 67.8811,Y 60.6155,Z 92,A 37.616,B 24.9068,C -2.2284,E1 25.1172,E2 47.318} C_DIS
LIN {X 65.4345,Y 63.2487,Z 92,A 39.2331,B 24.9084,C -2.2102,E1 25.1142,E2 45.7509} C_DIS
LIN {X 63.6182,Y 65.077,Z 92,A 41.173,B 24.9071,C -2.2249,E1 25.1102,E2 43.7844} C_DIS
LIN {X 60.8933,Y 67.6324,Z 92,A 43.3793,B 24.9071,C -2.2245,E1 25.1057,E2 41.588} C_DIS
LIN {X 57.7897,Y 70.304,Z 92,A 46.1511,B 24.9062,C -2.2362,E1 25.0997,E2 38.7991} C_DIS
LIN {X 51.6912,Y 74.9011,Z 92,A 50.4513,B 24.907,C -2.2267,E1 25.0902,E2 34.5368} C_DIS
LIN {X 48.399,Y 77.0691,Z 92,A 52.9909,B 24.9065,C -2.2326,E1 25.0842,E2 31.9915} C_DIS
LIN {X 45.4085,Y 78.8679,Z 92,A 55.2063,B 24.9062,C -2.2364,E1 25.0789,E2 29.7738} C_DIS
LIN {X 40.5775,Y 81.4589,Z 92,A 58.6855,B 24.9057,C -2.2419,E1 25.0703,E2 26.2915} C_DIS
LIN {X 37.5743,Y 82.8872,Z 92,A 60.7616,B 24.9056,C -2.2437,E1 25.065,E2 24.2163} C_DIS
LIN {X 35.3703,Y 83.8511,Z 92,A 62.4322,B 24.905,C -2.2507,E1 25.0607,E2 22.5331} C_DIS
LIN {X 29.8783,Y 85.9618,Z 92,A 65.6623,B 24.906,C -2.238,E1 25.0524,E2 19.3401} C_DIS
LIN {X 24.1516,Y 87.7437,Z 92,A 69.8729,B 24.9046,C -2.2555,E1 25.041,E2 15.0956} C_DIS
LIN {X 20.8164,Y 88.5938,Z 92,A 71.6754,B 24.9055,C -2.2444,E1 25.0362,E2 13.322} C_DIS
LIN {X 16.0231,Y 89.5842,Z 92,A 74.9716,B 24.9048,C -2.2529,E1 25.0271,E2 10.0095} C_DIS
LIN {X 12.7202,Y 90.1125,Z 92,A 77.0283,B 24.9048,C -2.2519,E1 25.0215,E2 7.9572} C_DIS
LIN {X 8.7069,Y 90.589,Z 92,A 79.4111,B 24.9053,C -2.2469,E1 25.0149,E2 5.5879} C_DIS
LIN {X 3.7103,Y 90.9304,Z 92,A 82.9071,B 24.9043,C -2.2582,E1 25.0051,E2 2.0664} C_DIS
LIN {X 0.1571,Y 91.0066,Z 92,A 85.1596,B 24.9043,C -2.2584,E1 24.9988,E2 -0.1862} C_DIS
LIN {X -3.6061,Y 90.9348,Z 92,A 87.8918,B 24.9034,C -2.2696,E1 24.9911,E2 -2.9455} C_DIS
LIN {X -6.8065,Y 90.7521,Z 92,A 89.5196,B 24.9045,C -2.2559,E1 24.9866,E2 -4.5414} C_DIS
LIN {X -10.0755,Y 90.4478,Z 92,A 91.3556,B 24.9053,C -2.2473,E1 24.9816,E2 -6.358} C_DIS
LIN {X -13.6589,Y 89.9753,Z 92,A 93.8115,B 24.9049,C -2.2517,E1 24.9748,E2 -8.8263} C_DIS
LIN {X -17.0608,Y 89.3925,Z 92,A 95.7343,B 24.9057,C -2.242,E1 24.9695,E2 -10.7279} C_DIS
LIN {X -20.8548,Y 88.5849,Z 92,A 99.0595,B 24.9035,C -2.2684,E1 24.9603,E2 -14.1201} C_DIS
LIN {X -24.4941,Y 87.6482,Z 92,A 100.7053,B 24.9056,C -2.2427,E1 24.956,E2 -15.7073} C_DIS
LIN {X -27.9143,Y 86.6191,Z 92,A 103.7293,B 24.9038,C -2.265,E1 24.9478,E2 -18.7899} C_DIS
LIN {X -31.6781,Y 85.3161,Z 92,A 105.3996,B 24.9063,C -2.235,E1 24.9436,E2 -20.3921} C_DIS
LIN {X -35.9825,Y 83.5913,Z 92,A 108.5094,B 24.9061,C -2.2369,E1 24.9356,E2 -23.5134} C_DIS
LIN {X -38.7609,Y 82.3396,Z 92,A 110.847,B 24.9053,C -2.2473,E1 24.9296,E2 -25.8816} C_DIS
LIN {X -44.2624,Y 79.5168,Z 92,A 114.4118,B 24.9067,C -2.2304,E1 24.9208,E2 -29.416} C_DIS
LIN {X -46.9112,Y 77.9845,Z 92,A 117.1601,B 24.9048,C -2.2528,E1 24.9141,E2 -32.2262} C_DIS
LIN {X -50.8239,Y 75.4921,Z 92,A 119.7092,B 24.9063,C -2.2354,E1 24.9083,E2 -34.7422} C_DIS
LIN {X -53.5685,Y 73.5699,Z 92,A 121.2704,B 24.9081,C -2.214,E1 24.9048,E2 -36.258} C_DIS
LIN {X -56.0653,Y 71.6866,Z 92,A 123.3086,B 24.9082,C -2.212,E1 24.9003,E2 -38.2987} C_DIS
LIN {X -60.3853,Y 68.0871,Z 92,A 126.979,B 24.9085,C -2.2081,E1 24.8925,E2 -41.9741} C_DIS
LIN {X -63.1245,Y 65.5543,Z 92,A 129.167,B 24.9094,C -2.1977,E1 24.8881,E2 -44.1462} C_DIS
LIN {X -65.5055,Y 63.1751,Z 92,A 131.3032,B 24.9098,C -2.1931,E1 24.8839,E2 -46.2806} C_DIS
LIN {X -67.7127,Y 60.8032,Z 92,A 133.9919,B 24.9086,C -2.2079,E1 24.8788,E2 -49.0166} C_DIS
LIN {X -70.0969,Y 58.0389,Z 92,A 135.7223,B 24.9105,C -2.1845,E1 24.8758,E2 -50.6992} C_DIS
LIN {X -72.2779,Y 55.2998,Z 92,A 138.1309,B 24.9105,C -2.1849,E1 24.8716,E2 -53.1201} C_DIS
LIN {X -74.6288,Y 52.083,Z 92,A 140.7259,B 24.9108,C -2.1807,E1 24.8674,E2 -55.7178} C_DIS
LIN {X -77.6671,Y 47.4334,Z 92,A 143.6125,B 24.9131,C -2.1524,E1 24.8632,E2 -58.5515} C_DIS
LIN {X -79.4212,Y 44.4336,Z 92,A 146.4522,B 24.912,C -2.1658,E1 24.8591,E2 -61.4379} C_DIS
LIN {X -81.1378,Y 41.2161,Z 92,A 148.3365,B 24.9136,C -2.1466,E1 24.8568,E2 -63.2865} C_DIS
LIN {X -82.9816,Y 37.3647,Z 92,A 150.834,B 24.9147,C -2.1329,E1 24.8538,E2 -65.7648} C_DIS
LIN {X -84.6188,Y 33.4929,Z 92,A 153.5189,B 24.9152,C -2.126,E1 24.8509,E2 -68.4481} C_DIS
LIN {X -86.6978,Y 27.6712,Z 92,A 157.8348,B 24.9152,C -2.1266,E1 24.8469,E2 -72.79} C_DIS
LIN {X -87.4892,Y 25.0552,Z 92,A 160.024,B 24.9145,C -2.1353,E1 24.8452,E2 -75.0127} C_DIS
LIN {X -88.3574,Y 21.7967,Z 92,A 162.0199,B 24.9153,C -2.1248,E1 24.8439,E2 -76.9951} C_DIS
LIN {X -89.3133,Y 17.4718,Z 92,A 164.4108,B 24.917,C -2.1039,E1 24.8425,E2 -79.3504} C_DIS
LIN {X -89.8586,Y 14.414,Z 92,A 166.2504,B 24.9178,C -2.0942,E1 24.8417,E2 -81.1777} C_DIS
LIN {X -90.2863,Y 11.4248,Z 92,A 168.3123,B 24.9178,C -2.0929,E1 24.8409,E2 -83.2489} C_DIS
LIN {X -90.6416,Y 8.137,Z 92,A 170.3662,B 24.9184,C -2.0854,E1 24.8403,E2 -85.2972} C_DIS
LIN {X -90.8017,Y 6.0922,Z 92,A 172.6426,B 24.9164,C -2.1111,E1 24.8399,E2 -87.6485} C_DIS
LIN {X -90.996,Y 1.3714,Z 92,A 174.7066,B 24.9193,C -2.0739,E1 24.8398,E2 -89.6363} C_DIS
LIN {X -90.9891,Y -1.7475,Z 92,A 176.643,B 24.9199,C -2.0669,E1 24.8398,E2 -91.5674} C_DIS
LIN {X -90.7622,Y -6.6765,Z 92,A 179.8615,B 24.9204,C -2.0603,E1 24.8403,E2 -94.7896} C_DIS
LIN {X -90.4757,Y -9.815,Z 92,A -178.0823,B 24.9207,C -2.0562,E1 24.8409,E2 -96.8484} C_DIS
LIN {X -90.025,Y -13.336,Z 92,A -175.9129,B 24.9214,C -2.0472,E1 24.8417,E2 -99.0091} C_DIS
LIN {X -89.5232,Y -16.3622,Z 92,A -173.9879,B 24.9219,C -2.041,E1 24.8427,E2 -100.9308} C_DIS
LIN {X -88.8841,Y -19.5374,Z 92,A -172.0569,B 24.9226,C -2.0314,E1 24.8438,E2 -102.8504} C_DIS
LIN {X -88.0949,Y -22.8339,Z 92,A -169.3275,B 24.9217,C -2.043,E1 24.8457,E2 -105.6233} C_DIS
LIN {X -86.6687,Y -27.7609,Z 92,A -166.5377,B 24.9235,C -2.0199,E1 24.8479,E2 -108.3741} C_DIS
LIN {X -83.9011,Y -35.2516,Z 92,A -161.4965,B 24.9246,C -2.0056,E1 24.8529,E2 -113.4095} C_DIS
LIN {X -82.5684,Y -38.2695,Z 92,A -159.3609,B 24.9249,C -2.0015,E1 24.8553,E2 -115.5471} C_DIS
LIN {X -80.9718,Y -41.5411,Z 92,A -157.016,B 24.9252,C -1.9968,E1 24.8583,E2 -117.8933} C_DIS
LIN {X -79.8526,Y -43.6546,Z 92,A -155.1952,B 24.9248,C -2.0024,E1 24.8607,E2 -119.7371} C_DIS
LIN {X -77.4453,Y -47.7968,Z 92,A -152.1276,B 24.9253,C -1.996,E1 24.8652,E2 -122.8053} C_DIS
LIN {X -75.0439,Y -51.4859,Z 92,A -149.7743,B 24.9268,C -1.976,E1 24.8688,E2 -125.1227} C_DIS
LIN {X -73.1433,Y -54.1512,Z 92,A -147.3522,B 24.9263,C -1.9822,E1 24.8728,E2 -127.5712} C_DIS
LIN {X -70.6482,Y -57.3664,Z 92,A -143.8258,B 24.9245,C -2.0066,E1 24.8792,E2 -131.1722} C_DIS
LIN {X -66.7816,Y -61.8259,Z 92,A -141.3698,B 24.9281,C -1.9584,E1 24.8836,E2 -133.5244} C_DIS
LIN {X -64.689,Y -64.0109,Z 92,A -138.242,B 24.9255,C -1.9932,E1 24.8899,E2 -136.7482} C_DIS
LIN {X -60.586,Y -67.9075,Z 92,A -135.7696,B 24.9286,C -1.9513,E1 24.8948,E2 -139.1309} C_DIS
LIN {X -56.4487,Y -71.3836,Z 92,A -132.1306,B 24.9286,C -1.9525,E1 24.9027,E2 -142.7865} C_DIS
LIN {X -53.2598,Y -73.795,Z 92,A -129.4867,B 24.9286,C -1.9522,E1 24.9087,E2 -145.439} C_DIS
LIN {X -50.3175,Y -75.8306,Z 92,A -127.3014,B 24.929,C -1.9465,E1 24.9138,E2 -147.6179} C_DIS
LIN {X -47.2568,Y -77.7744,Z 92,A -124.6948,B 24.9284,C -1.9536,E1 24.92,E2 -150.2495} C_DIS
LIN {X -43.8546,Y -79.7441,Z 92,A -122.7261,B 24.9299,C -1.9338,E1 24.9247,E2 -152.1767} C_DIS
LIN {X -40.5755,Y -81.46,Z 92,A -120.5305,B 24.9304,C -1.9265,E1 24.9302,E2 -154.3609} C_DIS
LIN {X -38.056,Y -82.6677,Z 92,A -118.6635,B 24.9304,C -1.928,E1 24.9349,E2 -156.2362} C_DIS
LIN {X -32.5864,Y -84.9726,Z 92,A -113.8634,B 24.928,C -1.9594,E1 24.9476,E2 -161.1215} C_DIS
LIN {X -27.3121,Y -86.8116,Z 92,A -111.3319,B 24.9306,C -1.9239,E1 24.9541,E2 -163.5732} C_DIS
LIN {X -23.038,Y -88.0424,Z 92,A -107.9337,B 24.9293,C -1.9421,E1 24.9634,E2 -167.0198} C_DIS
LIN {X -18.9081,Y -89.0213,Z 92,A -106.0435,B 24.9313,C -1.9147,E1 24.9684,E2 -168.8473} C_DIS
LIN {X -15.9014,Y -89.6061,Z 92,A -104.0932,B 24.9313,C -1.9147,E1 24.9737,E2 -170.7998} C_DIS
LIN {X -11.4212,Y -90.2868,Z 92,A -101.4474,B 24.9318,C -1.9072,E1 24.981,E2 -173.4297} C_DIS
LIN {X -6.0278,Y -90.8061,Z 92,A -97.8655,B 24.9314,C -1.9127,E1 24.991,E2 -177.0265} C_DIS
LIN {X -0.8883,Y -91.0021,Z 92,A -94.7243,B 24.9316,C -1.9098,E1 24.9998,E2 -180.1612} C_DIS
LIN {X 0.5684,Y -90.9983,Z 92,A -93.2034,B 24.9301,C -1.9307,E1 25.0042,E2 -181.7316} C_DIS
Enddeposition()
LIN {X 0.5684,Y -90.9983,Z 92,A -93.2034,B 24.9301,C -1.9307,E1 25.0042,E2 -181.7316} C_DIS
Startdeposition()
$VEL.CP = VEL_PRINT
LIN {X -1.1556,Y -90.0438,Z 92,A -95.8099,B 24.9326,C -1.8962,E1 24.9967,E2 -179.0434} C_DIS
LIN {X -4.6389,Y -89.9308,Z 92,A -97.9441,B 24.9324,C -1.8988,E1 24.9907,E2 -176.9147} C_DIS
LIN {X -6.9477,Y -89.7817,Z 92,A -99.8474,B 24.9334,C -1.8847,E1 24.9853,E2 -174.9773} C_DIS
LIN {X -11.2417,Y -89.3459,Z 92,A -102.2623,B 24.9326,C -1.8958,E1 24.9787,E2 -172.5872} C_DIS
LIN {X -14.6344,Y -88.853,Z 92,A -104.3043,B 24.9323,C -1.9009,E1 24.9731,E2 -170.5555} C_DIS
LIN {X -17.533,Y -88.3279,Z 92,A -106.3861,B 24.9327,C -1.8949,E1 24.9673,E2 -168.4572} C_DIS
LIN {X -22.199,Y -87.271,Z 92,A -109.2817,B 24.9322,C -1.9013,E1 24.9595,E2 -165.5728} C_DIS
LIN {X -25.6485,Y -86.3199,Z 92,A -111.4914,B 24.932,C -1.9049,E1 24.9535,E2 -163.3682} C_DIS
LIN {X -30.4653,Y -84.7408,Z 92,A -114.8339,B 24.932,C -1.9038,E1 24.9447,E2 -160.0167} C_DIS
LIN {X -32.9217,Y -83.816,Z 92,A -116.7892,B 24.9326,C -1.8963,E1 24.9395,E2 -158.0395} C_DIS
LIN {X -37.214,Y -82.0009,Z 92,A -119.3973,B 24.9316,C -1.9108,E1 24.9329,E2 -155.4596} C_DIS
LIN {X -39.9375,Y -80.7091,Z 92,A -121.3103,B 24.9314,C -1.9132,E1 24.9281,E2 -153.5475} C_DIS
LIN {X -42.6505,Y -79.3095,Z 92,A -123.3568,B 24.9314,C -1.9124,E1 24.9231,E2 -151.4935} C_DIS
LIN {X -46.72,Y -76.9819,Z 92,A -125.8633,B 24.9301,C -1.9315,E1 24.9171,E2 -149.0249} C_DIS
LIN {X -49.0519,Y -75.519,Z 92,A -128.17,B 24.9311,C -1.9169,E1 24.9116,E2 -146.676} C_DIS
LIN {X -52.7933,Y -72.9526,Z 92,A -130.9396,B 24.9305,C -1.9253,E1 24.9052,E2 -143.9169} C_DIS
LIN {X -56.6246,Y -70.0188,Z 92,A -134.6058,B 24.9314,C -1.9126,E1 24.8971,E2 -140.2071} C_DIS
LIN {X -59.3026,Y -67.7656,Z 92,A -136.0228,B 24.9293,C -1.9416,E1 24.8942,E2 -138.8535} C_DIS
LIN {X -62.2491,Y -65.0701,Z 92,A -139.2685,B 24.9305,C -1.9253,E1 24.8875,E2 -135.5557} C_DIS
LIN {X -65.7461,Y -61.5343,Z 92,A -142.4007,B 24.9299,C -1.9331,E1 24.8815,E2 -132.4285} C_DIS
LIN {X -69.7327,Y -56.9776,Z 92,A -145.8763,B 24.9285,C -1.9532,E1 24.8752,E2 -128.9851} C_DIS
LIN {X -73.4236,Y -52.1343,Z 92,A -149.8589,B 24.928,C -1.9594,E1 24.8686,E2 -124.9981} C_DIS
LIN {X -75.3443,Y -49.3183,Z 92,A -152.1475,B 24.9279,C -1.9614,E1 24.865,E2 -122.7027} C_DIS
LIN {X -76.831,Y -46.9682,Z 92,A -154.1271,B 24.9279,C -1.9597,E1 24.8621,E2 -120.709} C_DIS
LIN {X -79.3666,Y -42.5453,Z 92,A -157.0896,B 24.9267,C -1.9768,E1 24.8581,E2 -117.7717} C_DIS
LIN {X -81.0013,Y -39.3433,Z 92,A -159.3183,B 24.9261,C -1.9849,E1 24.8553,E2 -115.5502} C_DIS
LIN {X -82.3902,Y -36.3451,Z 92,A -161.4117,B 24.9257,C -1.9911,E1 24.8529,E2 -113.4601} C_DIS
LIN {X -84.6876,Y -30.6112,Z 92,A -165.3719,B 24.9249,C -2.0016,E1 24.8489,E2 -109.5029} C_DIS
LIN {X -85.7462,Y -27.5063,Z 92,A -167.3048,B 24.9241,C -2.0123,E1 24.8472,E2 -107.5845} C_DIS
LIN {X -86.9991,Y -23.2417,Z 92,A -170.2055,B 24.9236,C -2.0187,E1 24.845,E2 -104.6823} C_DIS
LIN {X -88.0833,Y -18.7222,Z 92,A -173.4019,B 24.9234,C -2.0208,E1 24.843,E2 -101.472} C_DIS
LIN {X -88.7616,Y -15.1809,Z 92,A -175.6184,B 24.9227,C -2.0302,E1 24.8419,E2 -99.2649} C_DIS
LIN {X -89.2323,Y -12.1192,Z 92,A -177.662,B 24.9224,C -2.0342,E1 24.841,E2 -97.2188} C_DIS
LIN {X -89.6188,Y -8.8159,Z 92,A -179.8002,B 24.9219,C -2.0403,E1 24.8404,E2 -95.0821} C_DIS
LIN {X -89.844,Y -6.0841,Z 92,A 178.3335,B 24.9218,C -2.0423,E1 24.84,E2 -93.2095} C_DIS
LIN {X -90.0138,Y -2.5535,Z 92,A 176.3168,B 24.9207,C -2.0562,E1 24.8398,E2 -91.2139} C_DIS
LIN {X -90.0456,Y 0.9903,Z 92,A 174.0248,B 24.9202,C -2.0623,E1 24.8398,E2 -88.9226} C_DIS
LIN {X -89.8828,Y 5.5075,Z 92,A 170.9518,B 24.92,C -2.0658,E1 24.8402,E2 -85.8395} C_DIS
LIN {X -89.5959,Y 9.0366,Z 92,A 168.7861,B 24.9192,C -2.0756,E1 24.8407,E2 -83.6841} C_DIS
LIN {X -89.0806,Y 13.1783,Z 92,A 166.0155,B 24.9188,C -2.0808,E1 24.8418,E2 -80.9093} C_DIS
LIN {X -88.5629,Y 16.3008,Z 92,A 164.0775,B 24.9181,C -2.0894,E1 24.8427,E2 -78.9803} C_DIS
LIN {X -87.3803,Y 21.768,Z 92,A 160.4372,B 24.9174,C -2.0983,E1 24.845,E2 -75.3398} C_DIS
LIN {X -86.424,Y 25.2973,Z 92,A 158.1836,B 24.9167,C -2.1077,E1 24.8467,E2 -73.0957} C_DIS
LIN {X -85.4073,Y 28.5413,Z 92,A 156.3085,B 24.9155,C -2.1228,E1 24.8482,E2 -71.246} C_DIS
LIN {X -83.805,Y 32.9497,Z 92,A 153.1391,B 24.9152,C -2.1266,E1 24.8513,E2 -68.0676} C_DIS
LIN {X -82.3691,Y 36.3935,Z 92,A 150.8464,B 24.9144,C -2.1361,E1 24.8538,E2 -65.785} C_DIS
LIN {X -80.463,Y 40.4341,Z 92,A 147.8622,B 24.9141,C -2.1404,E1 24.8574,E2 -62.7948} C_DIS
LIN {X -78.416,Y 44.2723,Z 92,A 144.8757,B 24.9139,C -2.142,E1 24.8614,E2 -59.7964} C_DIS
LIN {X -76.5939,Y 47.3552,Z 92,A 142.1032,B 24.9146,C -2.1341,E1 24.8655,E2 -56.9908} C_DIS
LIN {X -74.7104,Y 50.2731,Z 92,A 140.6113,B 24.9124,C -2.1612,E1 24.8677,E2 -55.5561} C_DIS
LIN {X -71.2035,Y 55.1277,Z 92,A 136.5336,B 24.9122,C -2.1636,E1 24.8745,E2 -51.4644} C_DIS
LIN {X -68.6957,Y 58.2219,Z 92,A 133.3113,B 24.9133,C -2.15,E1 24.8803,E2 -48.1948} C_DIS
LIN {X -65.9107,Y 61.3592,Z 92,A 131.319,B 24.9111,C -2.1765,E1 24.884,E2 -46.257} C_DIS
LIN {X -63.5062,Y 63.8438,Z 92,A 129.1231,B 24.9107,C -2.182,E1 24.8883,E2 -44.0647} C_DIS
LIN {X -60.9856,Y 66.2551,Z 92,A 126.885,B 24.9103,C -2.1866,E1 24.8928,E2 -41.8284} C_DIS
LIN {X -58.039,Y 68.8504,Z 92,A 124.1039,B 24.9106,C -2.1838,E1 24.8987,E2 -39.0298} C_DIS
LIN {X -54.5998,Y 71.6103,Z 92,A 121.7505,B 24.9089,C -2.2033,E1 24.9038,E2 -36.7142} C_DIS
LIN {X -51.9239,Y 73.5728,Z 92,A 119.386,B 24.9092,C -2.1999,E1 24.9092,E2 -34.3336} C_DIS
LIN {X -47.215,Y 76.681,Z 92,A 115.7986,B 24.9086,C -2.2068,E1 24.9176,E2 -30.7509} C_DIS
LIN {X -45.035,Y 77.9798,Z 92,A 113.3183,B 24.9106,C -2.1836,E1 24.9238,E2 -28.2082} C_DIS
LIN {X -40.8496,Y 80.2515,Z 92,A 111.0676,B 24.9082,C -2.2121,E1 24.9292,E2 -26.019} C_DIS
LIN {X -37.7188,Y 81.7701,Z 92,A 109.1189,B 24.9072,C -2.2236,E1 24.9341,E2 -24.0928} C_DIS
LIN {X -35.2337,Y 82.8712,Z 92,A 106.9081,B 24.9083,C -2.2114,E1 24.9398,E2 -21.8477} C_DIS
LIN {X -31.6911,Y 84.2893,Z 92,A 103.6158,B 24.9102,C -2.1883,E1 24.9486,E2 -18.4937} C_DIS
LIN {X -26.3021,Y 86.1238,Z 92,A 101.1126,B 24.907,C -2.2267,E1 24.955,E2 -16.0773} C_DIS
LIN {X -21.2109,Y 87.5162,Z 92,A 97.324,B 24.9078,C -2.2167,E1 24.9654,E2 -12.2594} C_DIS
LIN {X -17.9955,Y 88.2334,Z 92,A 95.7039,B 24.9064,C -2.2333,E1 24.9697,E2 -10.6768} C_DIS
LIN {X -14.7357,Y 88.836,Z 92,A 93.8073,B 24.9057,C -2.2416,E1 24.9748,E2 -8.7979} C_DIS
LIN {X -11.6397,Y 89.2944,Z 92,A 91.6985,B 24.9059,C -2.2391,E1 24.9807,E2 -6.6817} C_DIS
LIN {X -8.8372,Y 89.6167,Z 92,A 89.6715,B 24.9065,C -2.2327,E1 24.9864,E2 -4.6383} C_DIS
LIN {X -6.1952,Y 89.8365,Z 92,A 88.0471,B 24.9063,C -2.2354,E1 24.9909,E2 -3.0197} C_DIS
LIN {X -1.5315,Y 90.0369,Z 92,A 85.0923,B 24.9061,C -2.2368,E1 24.9991,E2 -0.0677} C_DIS
LIN {X 1.8196,Y 90.0315,Z 92,A 82.9779,B 24.9061,C -2.2377,E1 25.005,E2 2.0444} C_DIS
LIN {X 4.7876,Y 89.9226,Z 92,A 80.8291,B 24.9068,C -2.2295,E1 25.0111,E2 4.2119} C_DIS
LIN {X 8.6423,Y 89.6349,Z 92,A 78.5036,B 24.9064,C -2.2336,E1 25.0175,E2 6.5265} C_DIS
LIN {X 12.1224,Y 89.2318,Z 92,A 76.2737,B 24.9064,C -2.2331,E1 25.0237,E2 8.7558} C_DIS
LIN {X 16.4568,Y 88.5348,Z 92,A 73.244,B 24.9072,C -2.2244,E1 25.0321,E2 11.8029} C_DIS
LIN {X 20.9461,Y 87.5808,Z 92,A 70.6587,B 24.9064,C -2.2338,E1 25.039,E2 14.3623} C_DIS
LIN {X 23.9323,Y 86.8126,Z 92,A 68.14,B 24.908,C -2.2143,E1 25.0459,E2 16.9232} C_DIS
LIN {X 27.5106,Y 85.7449,Z 92,A 66.3699,B 24.9065,C -2.2324,E1 25.0505,E2 18.6472} C_DIS
LIN {X 29.8914,Y 84.944,Z 92,A 64.4624,B 24.9075,C -2.2208,E1 25.0556,E2 20.5784} C_DIS
LIN {X 34.484,Y 83.1868,Z 92,A 61.5435,B 24.9072,C -2.2246,E1 25.0631,E2 23.4817} C_DIS
LIN {X 38.299,Y 81.5,Z 92,A 59.0751,B 24.9069,C -2.2278,E1 25.0694,E2 25.9364} C_DIS
LIN {X 41.0052,Y 80.1719,Z 92,A 56.849,B 24.908,C -2.215,E1 25.075,E2 28.1867} C_DIS
LIN {X 44.8128,Y 78.1075,Z 92,A 54.0674,B 24.9084,C -2.2103,E1 25.0818,E2 30.9712} C_DIS
LIN {X 48.1215,Y 76.1152,Z 92,A 51.7517,B 24.9083,C -2.2113,E1 25.0872,E2 33.2771} C_DIS
LIN {X 51.1763,Y 74.0947,Z 92,A 49.1199,B 24.9094,C -2.1973,E1 25.0934,E2 35.9331} C_DIS
LIN {X 53.8428,Y 72.1804,Z 92,A 47.1555,B 24.9094,C -2.1979,E1 25.0977,E2 37.8892} C_DIS
LIN {X 57.5161,Y 69.2883,Z 92,A 44.9392,B 24.9077,C -2.2184,E1 25.1025,E2 40.0487} C_DIS
LIN {X 60.4796,Y 66.7194,Z 92,A 41.9807,B 24.9094,C -2.1975,E1 25.1087,E2 43.0449} C_DIS
LIN {X 63.1076,Y 64.2375,Z 92,A 39.7852,B 24.9095,C -2.1963,E1 25.1131,E2 45.234} C_DIS
LIN {X 67.7473,Y 59.3235,Z 92,A 35.4461,B 24.9104,C -2.1854,E1 25.1214,E2 49.5798} C_DIS
LIN {X 69.8849,Y 56.7897,Z 92,A 33.3344,B 24.9108,C -2.1804,E1 25.1252,E2 51.6935} C_DIS
LIN {X 72.1576,Y 53.8731,Z 92,A 31.1135,B 24.9109,C -2.1793,E1 25.1289,E2 53.9065} C_DIS
LIN {X 73.4399,Y 52.1114,Z 92,A 28.9581,B 24.9134,C -2.1491,E1 25.1325,E2 56.1229} C_DIS
LIN {X 75.7386,Y 48.7096,Z 92,A 26.7294,B 24.9128,C -2.1557,E1 25.1358,E2 58.3249} C_DIS
LIN {X 78.1415,Y 44.7537,Z 92,A 24.2491,B 24.9122,C -2.1642,E1 25.1393,E2 60.7723} C_DIS
LIN {X 79.9594,Y 41.421,Z 92,A 21.6516,B 24.9132,C -2.1511,E1 25.1427,E2 63.387} C_DIS
LIN {X 81.3841,Y 38.5466,Z 92,A 19.8869,B 24.9129,C -2.1552,E1 25.1449,E2 65.1326} C_DIS
LIN {X 82.9175,Y 35.1238,Z 92,A 16.653,B 24.9158,C -2.1185,E1 25.1485,E2 68.4354} C_DIS
LIN {X 84.411,Y 31.3654,Z 92,A 14.677,B 24.9147,C -2.132,E1 25.1504,E2 70.3684} C_DIS
LIN {X 86.3926,Y 25.4035,Z 92,A 10.9,B 24.9151,C -2.1279,E1 25.1537,E2 74.1337} C_DIS
LIN {X 87.222,Y 22.3896,Z 92,A 8.9423,B 24.9155,C -2.123,E1 25.1551,E2 76.0919} C_DIS
LIN {X 87.9198,Y 19.4721,Z 92,A 6.8452,B 24.9165,C -2.1104,E1 25.1564,E2 78.2065} C_DIS
LIN {X 88.7139,Y 15.4611,Z 92,A 4.4838,B 24.9165,C -2.1109,E1 25.1576,E2 80.553} C_DIS
LIN {X 89.2242,Y 12.176,Z 92,A 2.4605,B 24.9167,C -2.1075,E1 25.1584,E2 82.5723} C_DIS
LIN {X 89.6037,Y 8.9621,Z 92,A 0.3976,B 24.9172,C -2.1009,E1 25.1591,E2 84.6387} C_DIS
LIN {X 89.9879,Y 3.3741,Z 92,A -3.3811,B 24.9187,C -2.0818,E1 25.1597,E2 88.44} C_DIS
LIN {X 90.0245,Y -2.1806,Z 92,A -7.11,B 24.9202,C -2.0635,E1 25.1597,E2 92.1899} C_DIS
LIN {X 89.8336,Y -6.2388,Z 92,A -9.3373,B 24.9198,C -2.068,E1 25.1593,E2 94.3932} C_DIS
LIN {X 89.5519,Y -9.4565,Z 92,A -11.2307,B 24.9198,C -2.0672,E1 25.1588,E2 96.2772} C_DIS
LIN {X 89.1032,Y -13.0278,Z 92,A -13.743,B 24.921,C -2.0519,E1 25.1579,E2 98.8109} C_DIS
LIN {X 88.6028,Y -16.0788,Z 92,A -15.5931,B 24.9212,C -2.0498,E1 25.157,E2 100.6551} C_DIS
LIN {X 88.1788,Y -18.2619,Z 92,A -17.2713,B 24.9223,C -2.0359,E1 25.1561,E2 102.3564} C_DIS
LIN {X 86.888,Y -23.653,Z 92,A -20.7724,B 24.9231,C -2.0256,E1 25.1537,E2 105.8614} C_DIS
LIN {X 85.8962,Y -27.0362,Z 92,A -23.8917,B 24.9259,C -1.9875,E1 25.151,E2 109.053} C_DIS
LIN {X 84.1331,Y -32.1034,Z 92,A -26.0491,B 24.9234,C -2.0216,E1 25.149,E2 111.1178} C_DIS
LIN {X 82.4936,Y -36.108,Z 92,A -28.933,B 24.9244,C -2.0086,E1 25.1459,E2 114.0167} C_DIS
LIN {X 81.1987,Y -38.9325,Z 92,A -30.8594,B 24.9247,C -2.0045,E1 25.1436,E2 115.9424} C_DIS
LIN {X 79.5156,Y -42.2653,Z 92,A -33.0991,B 24.9248,C -2.0023,E1 25.1407,E2 118.1753} C_DIS
LIN {X 77.121,Y -46.491,Z 92,A -36.2952,B 24.9258,C -1.9896,E1 25.1363,E2 121.385} C_DIS
LIN {X 75.4102,Y -49.2184,Z 92,A -38.3548,B 24.9262,C -1.9834,E1 25.1331,E2 123.4488} C_DIS
LIN {X 73.7585,Y -51.6599,Z 92,A -40.2063,B 24.9266,C -1.979,E1 25.1302,E2 125.3014} C_DIS
LIN {X 71.7545,Y -54.4097,Z 92,A -42.1702,B 24.9265,C -1.9803,E1 25.127,E2 127.2529} C_DIS
LIN {X 70.245,Y -56.3454,Z 92,A -44.19,B 24.928,C -1.9599,E1 25.1234,E2 129.3114} C_DIS
LIN {X 67.5671,Y -59.5298,Z 92,A -46.5872,B 24.9278,C -1.962,E1 25.119,E2 131.693} C_DIS
LIN {X 65.3218,Y -61.9854,Z 92,A -48.4887,B 24.9277,C -1.9643,E1 25.1155,E2 133.5806} C_DIS
LIN {X 63.1923,Y -64.1538,Z 92,A -50.811,B 24.929,C -1.9459,E1 25.1108,E2 135.9365} C_DIS
LIN {X 60.1766,Y -66.9908,Z 92,A -53.1798,B 24.9288,C -1.9491,E1 25.106,E2 138.2883} C_DIS
LIN {X 57.6685,Y -69.1616,Z 92,A -55.278,B 24.9291,C -1.9447,E1 25.1015,E2 140.3885} C_DIS
LIN {X 54.8102,Y -71.4482,Z 92,A -57.7494,B 24.9298,C -1.9347,E1 25.096,E2 142.8744} C_DIS
LIN {X 51.8319,Y -73.6389,Z 92,A -60.1067,B 24.9302,C -1.9297,E1 25.0907,E2 145.2354} C_DIS
LIN {X 48.7702,Y -75.6998,Z 92,A -62.251,B 24.93,C -1.9322,E1 25.0857,E2 147.3666} C_DIS
LIN {X 46.1228,Y -77.3419,Z 92,A -64.693,B 24.9314,C -1.9126,E1 25.0798,E2 149.8472} C_DIS
LIN {X 42.5806,Y -79.3474,Z 92,A -67.3223,B 24.9318,C -1.9068,E1 25.0733,E2 152.4828} C_DIS
LIN {X 39.7338,Y -80.8101,Z 92,A -69.0916,B 24.9314,C -1.9126,E1 25.0689,E2 154.2336} C_DIS
LIN {X 36.0806,Y -82.5055,Z 92,A -71.4292,B 24.9311,C -1.9164,E1 25.063,E2 156.5564} C_DIS
LIN {X 34.0254,Y -83.3741,Z 92,A -73.8358,B 24.9337,C -1.8809,E1 25.0566,E2 159.0415} C_DIS
LIN {X 29.3219,Y -85.1438,Z 92,A -75.8779,B 24.9312,C -1.9158,E1 25.0515,E2 160.9968} C_DIS
LIN {X 23.1491,Y -87.0242,Z 92,A -80.1741,B 24.932,C -1.9047,E1 25.0399,E2 165.312} C_DIS
LIN {X 20.4721,Y -87.692,Z 92,A -81.9577,B 24.9322,C -1.9021,E1 25.0351,E2 167.0993} C_DIS
LIN {X 16.4761,Y -88.5313,Z 92,A -84.5233,B 24.9322,C -1.9009,E1 25.028,E2 169.6645} C_DIS
LIN {X 13.4143,Y -89.0457,Z 92,A -86.5155,B 24.9324,C -1.8989,E1 25.0225,E2 171.6595} C_DIS
LIN {X 8.8956,Y -89.6106,Z 92,A -89.4312,B 24.9326,C -1.8966,E1 25.0144,E2 174.5787} C_DIS
LIN {X 5.5741,Y -89.8785,Z 92,A -91.5561,B 24.9326,C -1.8955,E1 25.0085,E2 176.7052} C_DIS
LIN {X 1.227,Y -90.042,Z 92,A -94.4356,B 24.933,C -1.8909,E1 25.0004,E2 179.5949} C_DIS
LIN {X 1.227,Y -90.042,Z 92,A -94.4356,B 24.933,C -1.8909,E1 25.0004,E2 179.5949} C_DIS
Enddeposition()
LIN {X 0.5567,Y -89.0866,Z 92,A -93.9327,B 24.9296,C -1.9383,E1 25.0022,E2 178.9797} C_DIS
Startdeposition()
$VEL.CP = VEL_PRINT
LIN {X 4.252,Y -88.9932,Z 92,A -91.2743,B 24.9288,C -1.9483,E1 25.0096,E2 176.2982} C_DIS
LIN {X 7.587,Y -88.7714,Z 92,A -89.1569,B 24.9288,C -1.9483,E1 25.0155,E2 174.1819} C_DIS
LIN {X 10.8785,Y -88.4285,Z 92,A -87.0973,B 24.9289,C -1.9472,E1 25.0212,E2 172.1263} C_DIS
LIN {X 14.0817,Y -87.9751,Z 92,A -84.9035,B 24.9285,C -1.9525,E1 25.0273,E2 169.922} C_DIS
LIN {X 17.6835,Y -87.3215,Z 92,A -82.6237,B 24.9285,C -1.952,E1 25.0336,E2 167.6462} C_DIS
LIN {X 21.8358,Y -86.3772,Z 92,A -80.1903,B 24.9291,C -1.9443,E1 25.0401,E2 165.2345} C_DIS
LIN {X 28.6679,Y -84.3557,Z 92,A -75.2799,B 24.9279,C -1.9607,E1 25.0533,E2 160.2938} C_DIS
LIN {X 33.378,Y -82.6054,Z 92,A -72.4712,B 24.9287,C -1.9506,E1 25.0606,E2 157.5152} C_DIS
LIN {X 35.5077,Y -81.7123,Z 92,A -70.7103,B 24.9278,C -1.9622,E1 25.0652,E2 155.7309} C_DIS
LIN {X 38.2248,Y -80.4781,Z 92,A -68.6201,B 24.9272,C -1.9711,E1 25.0705,E2 153.6249} C_DIS
LIN {X 42.9047,Y -78.084,Z 92,A -65.1859,B 24.9266,C -1.9787,E1 25.079,E2 150.1825} C_DIS
LIN {X 46.365,Y -76.0788,Z 92,A -62.7502,B 24.9266,C -1.9787,E1 25.0848,E2 147.7543} C_DIS
LIN {X 49.5344,Y -74.056,Z 92,A -60.2984,B 24.9262,C -1.9845,E1 25.0906,E2 145.2967} C_DIS
LIN {X 52.5319,Y -71.9591,Z 92,A -58.1179,B 24.9262,C -1.9834,E1 25.0955,E2 143.1266} C_DIS
LIN {X 55.1388,Y -69.9816,Z 92,A -55.9792,B 24.9258,C -1.9891,E1 25.1002,E2 140.9823} C_DIS
LIN {X 57.7606,Y -67.8337,Z 92,A -53.8767,B 24.9257,C -1.9912,E1 25.1047,E2 138.8828} C_DIS
LIN {X 60.0565,Y -65.8101,Z 92,A -51.7981,B 24.925,C -1.9996,E1 25.1091,E2 136.7926} C_DIS
LIN {X 62.7791,Y -63.2181,Z 92,A -49.59,B 24.9251,C -1.998,E1 25.1135,E2 134.5974} C_DIS
LIN {X 64.3925,Y -61.5745,Z 92,A -47.8915,B 24.9243,C -2.0094,E1 25.1168,E2 132.8795} C_DIS
LIN {X 66.7328,Y -59.0314,Z 92,A -45.647,B 24.9238,C -2.0158,E1 25.121,E2 130.6299} C_DIS
LIN {X 68.7321,Y -56.6895,Z 92,A -43.7981,B 24.9238,C -2.0163,E1 25.1243,E2 128.7883} C_DIS
LIN {X 70.4373,Y -54.5557,Z 92,A -41.9972,B 24.9233,C -2.0225,E1 25.1274,E2 126.981} C_DIS
LIN {X 72.6913,Y -51.5145,Z 92,A -39.5662,B 24.9228,C -2.029,E1 25.1314,E2 124.5464} C_DIS
LIN {X 74.6821,Y -48.5856,Z 92,A -37.5036,B 24.9229,C -2.0277,E1 25.1346,E2 122.4973} C_DIS
LIN {X 76.0733,Y -46.3742,Z 92,A -35.1429,B 24.9207,C -2.057,E1 25.1381,E2 120.0794} C_DIS
LIN {X 77.7885,Y -43.4354,Z 92,A -33.778,B 24.9224,C -2.0337,E1 25.1399,E2 118.7766} C_DIS
LIN {X 78.924,Y -41.3368,Z 92,A -32.0181,B 24.9215,C -2.0463,E1 25.1423,E2 116.9962} C_DIS
LIN {X 80.3027,Y -38.5897,Z 92,A -30.0714,B 24.9211,C -2.0511,E1 25.1446,E2 115.0485} C_DIS
LIN {X 81.5479,Y -35.885,Z 92,A -28.1241,B 24.9206,C -2.058,E1 25.1469,E2 113.0955} C_DIS
LIN {X 83.0268,Y -32.3159,Z 92,A -25.8569,B 24.9206,C -2.0578,E1 25.1493,E2 110.8414} C_DIS
LIN {X 83.7727,Y -30.3294,Z 92,A -24.3851,B 24.92,C -2.0659,E1 25.1507,E2 109.3587} C_DIS
LIN {X 85.1339,Y -26.2665,Z 92,A -21.6334,B 24.9193,C -2.0743,E1 25.1531,E2 106.6027} C_DIS
LIN {X 86.2947,Y -22.1566,Z 92,A -18.4856,B 24.9175,C -2.0975,E1 25.1554,E2 103.4183} C_DIS
LIN {X 87.2037,Y -18.2573,Z 92,A -16.5357,B 24.9186,C -2.0831,E1 25.1565,E2 101.5138} C_DIS
LIN {X 87.5588,Y -16.4707,Z 92,A -15.0472,B 24.9174,C -2.0982,E1 25.1573,E2 99.9981} C_DIS
LIN {X 88.1443,Y -12.9798,Z 92,A -12.7197,B 24.9167,C -2.1074,E1 25.1583,E2 97.6629} C_DIS
LIN {X 88.6079,Y -9.2917,Z 92,A -10.513,B 24.9167,C -2.1084,E1 25.1591,E2 95.4667} C_DIS
LIN {X 88.8793,Y -6.18,Z 92,A -8.4763,B 24.916,C -2.1159,E1 25.1595,E2 93.4245} C_DIS
LIN {X 89.045,Y -2.9551,Z 92,A -6.4646,B 24.9157,C -2.1202,E1 25.1597,E2 91.4145} C_DIS
LIN {X 89.0939,Y 0.2444,Z 92,A -4.2987,B 24.9149,C -2.1307,E1 25.1597,E2 89.2368} C_DIS
LIN {X 88.9978,Y 4.145,Z 92,A -1.9661,B 24.9147,C -2.1323,E1 25.1595,E2 86.9141} C_DIS
LIN {X 88.7536,Y 7.7875,Z 92,A 0.4547,B 24.9139,C -2.1424,E1 25.159,E2 84.4839} C_DIS
LIN {X 88.4535,Y 10.6658,Z 92,A 2.3546,B 24.9133,C -2.1497,E1 25.1584,E2 82.578} C_DIS
LIN {X 87.9703,Y 14.1129,Z 92,A 4.6112,B 24.9127,C -2.1574,E1 25.1575,E2 80.3166} C_DIS
LIN {X 87.3321,Y 17.6319,Z 92,A 6.8547,B 24.9123,C -2.1625,E1 25.1563,E2 78.0741} C_DIS
LIN {X 86.6941,Y 20.5447,Z 92,A 8.7457,B 24.9119,C -2.1674,E1 25.1551,E2 76.1824} C_DIS
LIN {X 85.8531,Y 23.8156,Z 92,A 10.9522,B 24.9112,C -2.1753,E1 25.1535,E2 73.9701} C_DIS
LIN {X 84.4798,Y 28.2998,Z 92,A 13.8109,B 24.911,C -2.1787,E1 25.1511,E2 71.1196} C_DIS
LIN {X 83.3895,Y 31.3674,Z 92,A 16.789,B 24.9078,C -2.2166,E1 25.1481,E2 68.0686} C_DIS
LIN {X 81.7273,Y 35.4733,Z 92,A 18.7017,B 24.9099,C -2.1912,E1 25.1461,E2 66.2264} C_DIS
LIN {X 80.8767,Y 37.3725,Z 92,A 20.1308,B 24.9094,C -2.1982,E1 25.1445,E2 64.7885} C_DIS
LIN {X 79.4263,Y 40.3634,Z 92,A 22.2582,B 24.9089,C -2.2038,E1 25.1418,E2 62.6593} C_DIS
LIN {X 78.021,Y 43.0191,Z 92,A 24.103,B 24.9087,C -2.2059,E1 25.1394,E2 60.8191} C_DIS
LIN {X 76.4747,Y 45.7111,Z 92,A 26.2036,B 24.908,C -2.2149,E1 25.1364,E2 58.7081} C_DIS
LIN {X 74.8013,Y 48.4001,Z 92,A 28.1073,B 24.908,C -2.2155,E1 25.1335,E2 56.8126} C_DIS
LIN {X 72.7502,Y 51.432,Z 92,A 30.262,B 24.908,C -2.2144,E1 25.1302,E2 54.671} C_DIS
LIN {X 70.6072,Y 54.3353,Z 92,A 32.8366,B 24.9068,C -2.229,E1 25.1258,E2 52.0742} C_DIS
LIN {X 68.251,Y 57.2685,Z 92,A 35.0647,B 24.9068,C -2.228,E1 25.1219,E2 49.8589} C_DIS
LIN {X 65.5896,Y 60.2968,Z 92,A 38.2772,B 24.9046,C -2.2555,E1 25.1158,E2 46.5956} C_DIS
LIN {X 62.7901,Y 63.2072,Z 92,A 40.3649,B 24.9056,C -2.2432,E1 25.1118,E2 44.5458} C_DIS
LIN {X 60.797,Y 65.127,Z 92,A 42.2274,B 24.905,C -2.2498,E1 25.108,E2 42.6755} C_DIS
LIN {X 56.6658,Y 68.7518,Z 92,A 46.355,B 24.9027,C -2.2771,E1 25.0991,E2 38.4992} C_DIS
LIN {X 53.6453,Y 71.133,Z 92,A 48.8026,B 24.9024,C -2.2806,E1 25.0936,E2 36.0522} C_DIS
LIN {X 50.5204,Y 73.3863,Z 92,A 50.6784,B 24.9038,C -2.264,E1 25.0894,E2 34.2222} C_DIS
LIN {X 47.5206,Y 75.3633,Z 92,A 53.0275,B 24.9034,C -2.2689,E1 25.0839,E2 31.869} C_DIS
LIN {X 44.2064,Y 77.3533,Z 92,A 55.2703,B 24.9038,C -2.2643,E1 25.0786,E2 29.6441} C_DIS
LIN {X 41.323,Y 78.9313,Z 92,A 57.5914,B 24.903,C -2.2741,E1 25.0728,E2 27.3063} C_DIS
LIN {X 38.0294,Y 80.571,Z 92,A 59.9483,B 24.9028,C -2.2767,E1 25.0669,E2 24.9496} C_DIS
LIN {X 34.7547,Y 82.0356,Z 92,A 62.1744,B 24.9028,C -2.2765,E1 25.0612,E2 22.7293} C_DIS
LIN {X 31.6402,Y 83.2863,Z 92,A 64.2555,B 24.9028,C -2.276,E1 25.0558,E2 20.6538} C_DIS
LIN {X 29.64,Y 84.019,Z 92,A 65.6635,B 24.9026,C -2.2785,E1 25.0521,E2 19.2428} C_DIS
LIN {X 26.4292,Y 85.0834,Z 92,A 67.8005,B 24.9026,C -2.279,E1 25.0464,E2 17.1088} C_DIS
LIN {X 23.1638,Y 86.0299,Z 92,A 70.5196,B 24.9009,C -2.2981,E1 25.039,E2 14.3486} C_DIS
LIN {X 20.0463,Y 86.8092,Z 92,A 72.1211,B 24.9021,C -2.2838,E1 25.0347,E2 12.7833} C_DIS
LIN {X 16.7614,Y 87.5029,Z 92,A 74.0128,B 24.9028,C -2.276,E1 25.0296,E2 10.9125} C_DIS
LIN {X 14.254,Y 87.9472,Z 92,A 75.7334,B 24.9025,C -2.2793,E1 25.0249,E2 9.186} C_DIS
LIN {X 11.5209,Y 88.3457,Z 92,A 77.5321,B 24.9025,C -2.2805,E1 25.0199,E2 7.386} C_DIS
LIN {X 8.5777,Y 88.6807,Z 92,A 79.591,B 24.902,C -2.2857,E1 25.0141,E2 5.316} C_DIS
LIN {X 5.627,Y 88.9167,Z 92,A 81.5212,B 24.902,C -2.2866,E1 25.0087,E2 3.3845} C_DIS
LIN {X 2.3883,Y 89.0624,Z 92,A 83.3932,B 24.9025,C -2.2796,E1 25.0036,E2 1.5297} C_DIS
LIN {X -0.2132,Y 89.0941,Z 92,A 85.2625,B 24.902,C -2.2856,E1 24.9983,E2 -0.3538} C_DIS
LIN {X -3.3537,Y 89.0318,Z 92,A 87.2821,B 24.902,C -2.285,E1 24.9927,E2 -2.3722} C_DIS
LIN {X -6.6504,Y 88.8463,Z 92,A 89.4422,B 24.902,C -2.2853,E1 24.9867,E2 -4.5338} C_DIS
LIN {X -10.1959,Y 88.5085,Z 92,A 91.721,B 24.9022,C -2.2837,E1 24.9803,E2 -6.8102} C_DIS
LIN {X -13.9681,Y 87.9927,Z 92,A 93.9365,B 24.9029,C -2.2748,E1 24.9743,E2 -9.0062} C_DIS
LIN {X -16.4432,Y 87.5641,Z 92,A 95.8043,B 24.9023,C -2.2815,E1 24.9691,E2 -10.8919} C_DIS
LIN {X -21.3639,Y 86.4947,Z 92,A 99.0037,B 24.9027,C -2.2773,E1 24.9604,E2 -14.0856} C_DIS
LIN {X -24.2458,Y 85.7312,Z 92,A 100.8175,B 24.9031,C -2.2721,E1 24.9555,E2 -15.8898} C_DIS
LIN {X -27.2861,Y 84.8126,Z 92,A 102.9643,B 24.9031,C -2.2731,E1 24.9498,E2 -18.0425} C_DIS
LIN {X -31.7042,Y 83.262,Z 92,A 105.9539,B 24.9035,C -2.2686,E1 24.942,E2 -21.0275} C_DIS
LIN {X -35.109,Y 81.8862,Z 92,A 108.2053,B 24.904,C -2.2618,E1 24.9362,E2 -23.2678} C_DIS
LIN {X -37.6427,Y 80.751,Z 92,A 110.1728,B 24.9038,C -2.2647,E1 24.9311,E2 -25.2472} C_DIS
LIN {X -40.2399,Y 79.4893,Z 92,A 112.2881,B 24.9034,C -2.2697,E1 24.9258,E2 -27.3799} C_DIS
LIN {X -43.5182,Y 77.7423,Z 92,A 114.4431,B 24.9043,C -2.2584,E1 24.9206,E2 -29.5143} C_DIS
LIN {X -46.3796,Y 76.0699,Z 92,A 116.4677,B 24.9049,C -2.2513,E1 24.9158,E2 -31.5281} C_DIS
LIN {X -48.9799,Y 74.4222,Z 92,A 118.5458,B 24.9049,C -2.2506,E1 24.9109,E2 -33.6111} C_DIS
LIN {X -50.9728,Y 73.0718,Z 92,A 120.6715,B 24.9037,C -2.2651,E1 24.9059,E2 -35.7786} C_DIS
LIN {X -53.8801,Y 70.9566,Z 92,A 122.1807,B 24.9062,C -2.2359,E1 24.9027,E2 -37.2237} C_DIS
LIN {X -58.3284,Y 67.3471,Z 92,A 126.5617,B 24.9051,C -2.2488,E1 24.8932,E2 -41.6522} C_DIS
LIN {X -61.6635,Y 64.3067,Z 92,A 129.0239,B 24.9068,C -2.2288,E1 24.8882,E2 -44.0768} C_DIS
LIN {X -64.0824,Y 61.8962,Z 92,A 131.1688,B 24.9074,C -2.222,E1 24.884,E2 -46.2145} C_DIS
LIN {X -67.4793,Y 58.1765,Z 92,A 135.1139,B 24.9063,C -2.2349,E1 24.8766,E2 -50.2081} C_DIS
LIN {X -69.766,Y 55.4115,Z 92,A 136.4671,B 24.9092,C -2.2004,E1 24.8744,E2 -51.4855} C_DIS
LIN {X -72.5287,Y 51.7424,Z 92,A 140.0455,B 24.9083,C -2.211,E1 24.8684,E2 -55.1062} C_DIS
LIN {X -75.3311,Y 47.5721,Z 92,A 143.139,B 24.9094,C -2.1979,E1 24.8637,E2 -58.184} C_DIS
LIN {X -77.0663,Y 44.7059,Z 92,A 145.188,B 24.9102,C -2.1886,E1 24.8608,E2 -60.2215} C_DIS
LIN {X -78.8157,Y 41.5425,Z 92,A 147.3685,B 24.9111,C -2.1776,E1 24.8579,E2 -62.3873} C_DIS
LIN {X -81.3786,Y 36.2678,Z 92,A 151.0933,B 24.9121,C -2.165,E1 24.8534,E2 -66.1022} C_DIS
LIN {X -82.7991,Y 32.8956,Z 92,A 153.8654,B 24.9117,C -2.1701,E1 24.8504,E2 -68.9018} C_DIS
LIN {X -84.2546,Y 28.9678,Z 92,A 156.4924,B 24.9125,C -2.1598,E1 24.848,E2 -71.5193} C_DIS
LIN {X -85.1775,Y 26.126,Z 92,A 158.4316,B 24.9129,C -2.1544,E1 24.8464,E2 -73.4566} C_DIS
LIN {X -86.0733,Y 23.003,Z 92,A 160.4525,B 24.9136,C -2.1458,E1 24.8449,E2 -75.4688} C_DIS
LIN {X -86.8645,Y 19.8069,Z 92,A 162.8316,B 24.9136,C -2.1468,E1 24.8433,E2 -77.8641} C_DIS
LIN {X -87.5482,Y 16.5261,Z 92,A 164.7532,B 24.9147,C -2.1331,E1 24.8423,E2 -79.7644} C_DIS
LIN {X -88.3372,Y 11.5864,Z 92,A 167.8338,B 24.9158,C -2.1188,E1 24.841,E2 -82.8294} C_DIS
LIN {X -88.6553,Y 8.8384,Z 92,A 169.812,B 24.9158,C -2.1189,E1 24.8404,E2 -84.8196} C_DIS
LIN {X -88.9188,Y 5.5951,Z 92,A 172.0995,B 24.9158,C -2.1179,E1 24.84,E2 -87.1184} C_DIS
LIN {X -89.0602,Y 2.4604,Z 92,A 173.989,B 24.9167,C -2.1077,E1 24.8398,E2 -88.995} C_DIS
LIN {X -89.0884,Y -1.1077,Z 92,A 176.3541,B 24.9171,C -2.1024,E1 24.8398,E2 -91.3616} C_DIS
LIN {X -88.977,Y -4.5714,Z 92,A 178.5825,B 24.9177,C -2.0953,E1 24.8401,E2 -93.5865} C_DIS
LIN {X -88.7163,Y -8.1918,Z 92,A -179.0872,B 24.9183,C -2.0878,E1 24.8406,E2 -95.9128} C_DIS
LIN {X -88.3722,Y -11.3163,Z 92,A -177.1368,B 24.9189,C -2.0793,E1 24.8413,E2 -97.8547} C_DIS
LIN {X -87.9779,Y -14.0638,Z 92,A -175.1787,B 24.9189,C -2.0788,E1 24.8421,E2 -99.8232} C_DIS
LIN {X -87.2927,Y -17.8238,Z 92,A -172.5356,B 24.9191,C -2.0767,E1 24.8435,E2 -102.4769} C_DIS
LIN {X -86.4544,Y -21.5294,Z 92,A -170.3112,B 24.9202,C -2.0627,E1 24.845,E2 -104.6809} C_DIS
LIN {X -85.3287,Y -25.6281,Z 92,A -167.701,B 24.9211,C -2.0508,E1 24.847,E2 -107.2779} C_DIS
LIN {X -84.3929,Y -28.5576,Z 92,A -165.6258,B 24.9214,C -2.0478,E1 24.8488,E2 -109.3579} C_DIS
LIN {X -83.3043,Y -31.5924,Z 92,A -163.3366,B 24.9214,C -2.0482,E1 24.851,E2 -111.6608} C_DIS
LIN {X -81.7561,Y -35.4073,Z 92,A -160.8685,B 24.9223,C -2.0352,E1 24.8537,E2 -114.1117} C_DIS
LIN {X -80.3142,Y -38.5657,Z 92,A -158.6361,B 24.9228,C -2.0289,E1 24.8563,E2 -116.3413} C_DIS
LIN {X -78.8946,Y -41.3926,Z 92,A -156.6024,B 24.9232,C -2.0233,E1 24.8589,E2 -118.3725} C_DIS
LIN {X -75.9349,Y -46.6019,Z 92,A -152.9034,B 24.9244,C -2.0084,E1 24.8641,E2 -122.0551} C_DIS
LIN {X -74.4939,Y -48.8712,Z 92,A -150.9474,B 24.9242,C -2.0108,E1 24.867,E2 -124.0267} C_DIS
LIN {X -72.466,Y -51.8303,Z 92,A -148.4142,B 24.9242,C -2.0119,E1 24.8711,E2 -126.575} C_DIS
LIN {X -69.7504,Y -55.4313,Z 92,A -145.6773,B 24.925,C -2,E1 24.8758,E2 -129.2964} C_DIS
LIN {X -67.4814,Y -58.1741,Z 92,A -143.319,B 24.9252,C -1.9968,E1 24.88,E2 -131.6579} C_DIS
LIN {X -64.4231,Y -61.5427,Z 92,A -140.0934,B 24.925,C -1.9996,E1 24.8862,E2 -134.9043} C_DIS
LIN {X -59.3327,Y -66.4631,Z 92,A -136.1916,B 24.9272,C -1.9703,E1 24.894,E2 -138.7523} C_DIS
LIN {X -57.4465,Y -68.1013,Z 92,A -134.2339,B 24.9266,C -1.978,E1 24.8982,E2 -140.7359} C_DIS
LIN {X -53.2082,Y -71.4614,Z 92,A -131.1806,B 24.9281,C -1.9586,E1 24.9049,E2 -143.7544} C_DIS
LIN {X -50.2249,Y -73.5884,Z 92,A -128.4773,B 24.9276,C -1.9654,E1 24.9111,E2 -146.4832} C_DIS
LIN {X -47.6582,Y -75.277,Z 92,A -126.4385,B 24.9276,C -1.9643,E1 24.9159,E2 -148.5259} C_DIS
LIN {X -44.8019,Y -77.0111,Z 92,A -124.252,B 24.9278,C -1.9624,E1 24.9212,E2 -150.7146} C_DIS
LIN {X -41.7339,Y -78.7149,Z 92,A -122.0155,B 24.9281,C -1.9588,E1 24.9266,E2 -152.9488} C_DIS
LIN {X -39.2996,Y -79.9583,Z 92,A -120.2121,B 24.9281,C -1.9581,E1 24.9312,E2 -154.7553} C_DIS
LIN {X -36.117,Y -81.4465,Z 92,A -118.1799,B 24.9288,C -1.9483,E1 24.9363,E2 -156.7693} C_DIS
LIN {X -33.3202,Y -82.6289,Z 92,A -116.3357,B 24.9292,C -1.9429,E1 24.941,E2 -158.6047} C_DIS
LIN {X -30.0139,Y -83.8877,Z 92,A -113.7835,B 24.9287,C -1.9497,E1 24.9477,E2 -161.1783} C_DIS
LIN {X -26.6769,Y -85.0066,Z 92,A -111.8173,B 24.9296,C -1.9384,E1 24.9529,E2 -163.1213} C_DIS
LIN {X -23.1962,Y -86.0211,Z 92,A -109.6887,B 24.9301,C -1.9303,E1 24.9586,E2 -165.2343} C_DIS
LIN {X -21.2877,Y -86.5133,Z 92,A -107.9634,B 24.9291,C -1.9443,E1 24.9633,E2 -166.9952} C_DIS
LIN {X -19.1004,Y -87.0223,Z 92,A -106.4801,B 24.9291,C -1.9449,E1 24.9674,E2 -168.4818} C_DIS
LIN {X -16.4282,Y -87.567,Z 92,A -104.8822,B 24.9295,C -1.9391,E1 24.9717,E2 -170.0678} C_DIS
LIN {X -13.851,Y -88.0108,Z 92,A -103.0009,B 24.9291,C -1.9452,E1 24.9769,E2 -171.9651} C_DIS
LIN {X -11.016,Y -88.4111,Z 92,A -101.1293,B 24.9291,C -1.9458,E1 24.9821,E2 -173.8397} C_DIS
LIN {X -7.7221,Y -88.7597,Z 92,A -99.2404,B 24.9296,C -1.9377,E1 24.9873,E2 -175.7103} C_DIS
LIN {X -5.4053,Y -88.9309,Z 92,A -97.4216,B 24.9288,C -1.9484,E1 24.9925,E2 -177.5552} C_DIS
LIN {X -1.7563,Y -89.0765,Z 92,A -95.2418,B 24.9292,C -1.9432,E1 24.9985,E2 -179.7229} C_DIS
LIN {X 0.5567,Y -89.0866,Z 92,A -93.9315,B 24.9296,C -1.9378,E1 25.0022,E2 -181.0203} C_DIS
Enddeposition()
LIN {X 0.5567,Y -89.0866,Z 92,A -93.9315,B 24.9296,C -1.9378,E1 25.0022,E2 -181.0203} C_DIS
Startdeposition()
$VEL.CP = VEL_PRINT
LIN {X -1.0953,Y -88.1324,Z 92,A -95.7315,B 24.9301,C -1.9304,E1 24.9971,E2 -179.2029} C_DIS
LIN {X -3.251,Y -88.0793,Z 92,A -97.2612,B 24.9304,C -1.9261,E1 24.9928,E2 -177.6628} C_DIS
LIN {X -6.6065,Y -87.8907,Z 92,A -99.4084,B 24.9304,C -1.9273,E1 24.9868,E2 -175.5176} C_DIS
LIN {X -9.7185,Y -87.6019,Z 92,A -101.3338,B 24.9301,C -1.9309,E1 24.9815,E2 -173.5995} C_DIS
LIN {X -11.9956,Y -87.3185,Z 92,A -102.7517,B 24.9299,C -1.9335,E1 24.9776,E2 -172.1868} C_DIS
LIN {X -14.131,Y -86.9984,Z 92,A -104.08,B 24.9297,C -1.9363,E1 24.9739,E2 -170.8639} C_DIS
LIN {X -16.1342,Y -86.65,Z 92,A -105.5473,B 24.93,C -1.9321,E1 24.9698,E2 -169.3853} C_DIS
LIN {X -18.3754,Y -86.2019,Z 92,A -107.0948,B 24.9301,C -1.9308,E1 24.9656,E2 -167.8329} C_DIS
LIN {X -21.4216,Y -85.4965,Z 92,A -109.1435,B 24.9301,C -1.9314,E1 24.96,E2 -165.7827} C_DIS
LIN {X -24.5022,Y -84.6648,Z 92,A -111.1411,B 24.9298,C -1.9351,E1 24.9547,E2 -163.7908} C_DIS
LIN {X -26.7571,Y -83.9789,Z 92,A -112.5368,B 24.9294,C -1.9405,E1 24.951,E2 -162.4055} C_DIS
LIN {X -28.6832,Y -83.3415,Z 92,A -114.001,B 24.9297,C -1.937,E1 24.9471,E2 -160.9303} C_DIS
LIN {X -30.8301,Y -82.5707,Z 92,A -115.3431,B 24.9292,C -1.9427,E1 24.9436,E2 -159.599} C_DIS
LIN {X -32.8399,Y -81.7922,Z 92,A -116.7601,B 24.9292,C -1.9435,E1 24.9399,E2 -158.1809} C_DIS
LIN {X -34.8512,Y -80.9556,Z 92,A -118.2435,B 24.9292,C -1.9429,E1 24.9361,E2 -156.6926} C_DIS
LIN {X -36.7096,Y -80.1308,Z 92,A -119.7658,B 24.9296,C -1.9382,E1 24.9322,E2 -155.1554} C_DIS
LIN {X -39.629,Y -78.7279,Z 92,A -121.6803,B 24.929,C -1.9466,E1 24.9274,E2 -153.2559} C_DIS
LIN {X -41.6567,Y -77.6733,Z 92,A -123.1697,B 24.9288,C -1.9484,E1 24.9237,E2 -151.7666} C_DIS
LIN {X -43.547,Y -76.6295,Z 92,A -124.7453,B 24.9291,C -1.9451,E1 24.9199,E2 -150.1786} C_DIS
LIN {X -46.2464,Y -75.032,Z 92,A -126.6906,B 24.9286,C -1.9509,E1 24.9152,E2 -148.2411} C_DIS
LIN {X -48.1733,Y -73.8088,Z 92,A -128.1115,B 24.9283,C -1.9551,E1 24.9119,E2 -146.8256} C_DIS
LIN {X -50.3024,Y -72.3734,Z 92,A -129.9012,B 24.9284,C -1.9542,E1 24.9078,E2 -145.0278} C_DIS
LIN {X -52.6378,Y -70.694,Z 92,A -131.8321,B 24.9284,C -1.9555,E1 24.9034,E2 -143.0933} C_DIS
Enddeposition()
END
